PH_3302_08_ONN W153.07 BOOL  ; PH. MB FEED IN CONFIRM on
PH_3302_09_OFF W154.09 BOOL  ; PH. WORK FULL off
PH_3302_09_ON W151.09 BOOL  ; PH. WORK FULL on
PH_3302_10_OFF W154.10 BOOL  ; PH.TRANSFER STATION DIAPH SIDE CONFIRM off
PH_3302_10_ON W151.10 BOOL  ; PH.TRANSFER STATION DIAPH SIDE CONFIRM on
PH_3302_11_OFF W154.11 BOOL  ; PH.TRANSFER STATION DIAPH WORK CONFIRM off
PH_3302_11_ON W151.11 BOOL  ; PH.TRANSFER STATION DIAPH WORK CONFIRM on
PH_3302_12_OFF W154.12 BOOL  ; PH.TRANSFER STATION M&B WORK CONFIRM off
PH_3302_12_ON W151.12 BOOL  ; PH.TRANSFER STATION M&B WORK CONFIRM on
PH_3302_13_OFF W154.13 BOOL  ; PH. M&B LOADER WORK CONF 1 off
PH_3302_13_ON W151.13 BOOL  ; PH. M&B LOADER WORK CONF 1 on
PH_3302_14_OFF W154.14 BOOL  ; PH. M&B LOADER WORK CONF 2 off
PH_3302_14_ON W151.14 BOOL  ; PH. M&B LOADER WORK CONF 2 on
PH_3302_15_OFF W154.15 BOOL  ; PH. WORK IN ROTATE UNIT CONFIRM off
PH_3302_15_ON W151.15 BOOL  ; PH. WORK IN ROTATE UNIT CONFIRM on
PH_3304_08_OFF W156.08 BOOL  ; PH. WORK ROTATE PRE-END CONFIRM of
PH_3304_08_ON W153.08 BOOL  ; PH. WORK ROTATE PRE-END CONFIRM on
PH_3304_09_OFF W156.09 BOOL  ; PH. TEMINAL IN POSITION CONFIRM off
PH_3304_09_ON W153.09 BOOL  ; PH. TEMINAL IN POSITION CONFIRM on
PH_3304_10_OFF W156.10 BOOL  ; PH. WORK DIAPH LOAD IN CONFIRM off
PH_3304_10_ON W153.10 BOOL  ; PH. WORK DIAPH LOAD IN CONFIRM on
PH_3304_11_OFF W156.11 BOOL  ; PH.STATION DIAPH VACCUM CONFIRM off
PH_3304_11_ON W153.11 BOOL  ; PH.STATION DIAPH VACCUM CONFIRM on
PH_3304_12_OFF W156.12 BOOL  ; PH.STATION BUFFER DIAPH CONFIRM off
PH_3304_12_ON W153.12 BOOL  ; PH.STATION BUFFER DIAPH CONFIRM on
PH_3304_13_OFF W156.13 BOOL  ; PH. WORK NG CONFIRM off
PH_3304_13_ON W153.13 BOOL  ; PH. WORK NG CONFIRM on
PH_3304_14_OFF W156.14 BOOL  ; PH. WORK OK CONFIRM off
PH_3304_14_ON W153.14 BOOL  ; PH. WORK OK CONFIRM on
PRESSURE_NORMAL W100.01 BOOL  ; AIR SOURCE CONFIRM.
PSD W509 WORD[3]  ; SystemArea
SAFETY_DOOR W100.08 BOOL  ; CR.MACHINR DOOR CONFIRM
SHUTTER_DOOR_IN W100.11 BOOL  ; CR.SHUTTER DOOR IN CONFIRM
SHUTTER_DOOR_OUT W100.10 BOOL  ; CR.SHUTTER DOOR OUT CONFIRM
SS_AUTO W100.02 BOOL  ; AUTO.IND.(AUTO=on) On
SS_IND W200.02 BOOL  ; AUTO.IND.(AUTO=on) off
Stopwatch E0_4 UINT
Stopwatch_2 E0_5 UINT
TEACH_ON W100.07 BOOL  ; CR.TEACHING ON
sim_mch E0_3.10 BOOL

## Program P10_MAIN (cyclic task 0)
; STATION STATION CHECK
Local symbols
ALT36 T3042 TIMER
ALT37 T3000 TIMER
Disch_Command_P11 E0_3.11 BOOL
Disch_compl_aux E0_3.12 BOOL
Disch_compl_aux2 E0_3.13 BOOL
E0_3201_06 E0_46.04 BOOL  ; pin down
GB010_069 E0_3.14 BOOL  ; Homepos for discharge
Homepos_after_disch E0_3.15 BOOL
LB2341 E0_45.15 BOOL  ; PB trial mode
LB3421 E0_46.06 BOOL  ; GP1 takeout fault
LB523 E0_6.00 BOOL  ; Homeps 1 cond
LB5342 E0_45.14 BOOL  ; trigger ct
LB5431 E0_45.13 BOOL  ; trigger ct history
LD312 E0_48 UINT
LT028 T3033 TIMER
LT213 T3001 TIMER
LT214 T3002 TIMER
LT215 T3003 TIMER
LT216 T3004 TIMER
LT217 T3005 TIMER
LT2341 T3038 TIMER
LT321 T3006 TIMER  ; disch cancel
LT323 T3022 TIMER
LT324 T3021 TIMER
LT4014 T3007 TIMER
LT40505 T3008 TIMER
LT476 T3009 TIMER
LT567 T3031 TIMER
LT645 T3010 TIMER
LT765 T3034 TIMER  ; timeout positioning
LT976 T3011 TIMER
Machine_stop E0_6.01 BOOL
NOP E0_6.02 BOOL
Simulation_MCH E0_6.03 BOOL
disch_cancel E0_47.10 BOOL
nunggu_PSU E0_6.04 BOOL
rewrwe T3012 TIMER  ; Work On-> NG judge
tstt E0_45.12 BOOL

### Section MAIN

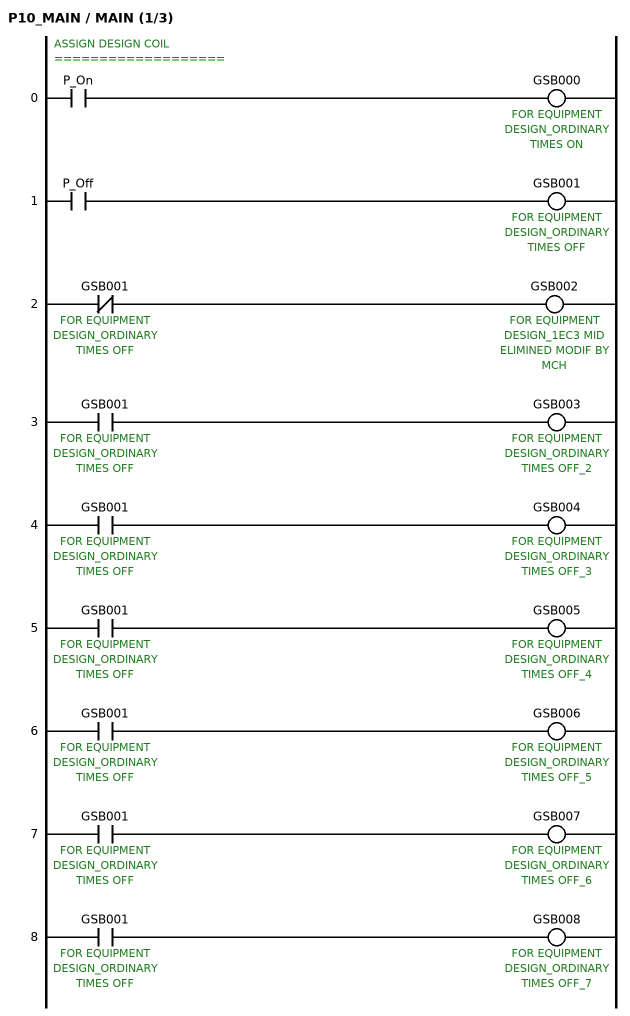
; rung 0: ASSIGN DESIGN COIL / ===================
LD P_On
OUT GSB000  ; FOR EQUIPMENT DESIGN_ORDINARY TIMES ON
; rung 1
LD P_Off
OUT GSB001  ; FOR EQUIPMENT DESIGN_ORDINARY TIMES OFF
; rung 2
LDNOT GSB001  ; FOR EQUIPMENT DESIGN_ORDINARY TIMES OFF
OUT GSB002  ; FOR EQUIPMENT DESIGN_1EC3 MID ELIMINED MODIF BY MCH
; rung 3
LD GSB001  ; FOR EQUIPMENT DESIGN_ORDINARY TIMES OFF
OUT GSB003  ; FOR EQUIPMENT DESIGN_ORDINARY TIMES OFF_2
; rung 4
LD GSB001  ; FOR EQUIPMENT DESIGN_ORDINARY TIMES OFF
OUT GSB004  ; FOR EQUIPMENT DESIGN_ORDINARY TIMES OFF_3
; rung 5
LD GSB001  ; FOR EQUIPMENT DESIGN_ORDINARY TIMES OFF
OUT GSB005  ; FOR EQUIPMENT DESIGN_ORDINARY TIMES OFF_4
; rung 6
LD GSB001  ; FOR EQUIPMENT DESIGN_ORDINARY TIMES OFF
OUT GSB006  ; FOR EQUIPMENT DESIGN_ORDINARY TIMES OFF_5
; rung 7
LD GSB001  ; FOR EQUIPMENT DESIGN_ORDINARY TIMES OFF
OUT GSB007  ; FOR EQUIPMENT DESIGN_ORDINARY TIMES OFF_6
; rung 8
LD GSB001  ; FOR EQUIPMENT DESIGN_ORDINARY TIMES OFF
OUT GSB008  ; FOR EQUIPMENT DESIGN_ORDINARY TIMES OFF_7

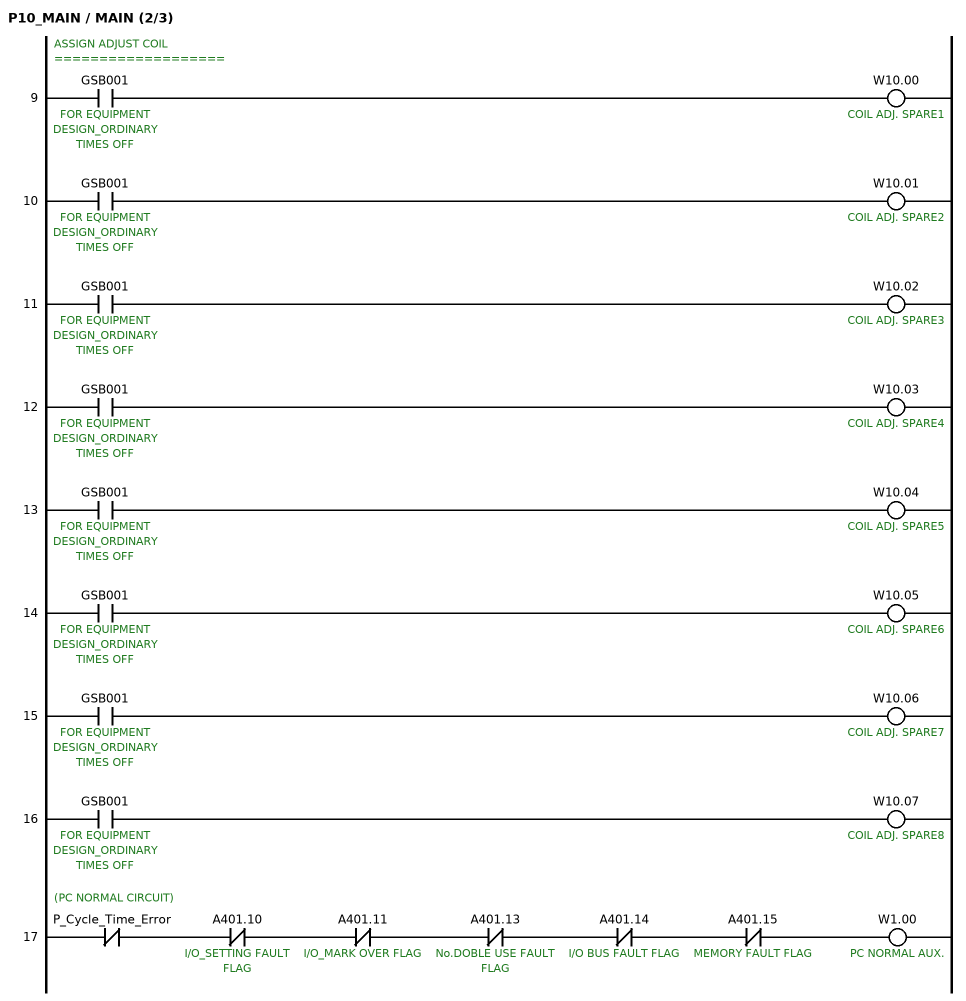
; rung 9: ASSIGN ADJUST COIL / ===================
LD GSB001  ; FOR EQUIPMENT DESIGN_ORDINARY TIMES OFF
OUT W10.00  ; COIL ADJ. SPARE1
; rung 10
LD GSB001  ; FOR EQUIPMENT DESIGN_ORDINARY TIMES OFF
OUT W10.01  ; COIL ADJ. SPARE2
; rung 11
LD GSB001  ; FOR EQUIPMENT DESIGN_ORDINARY TIMES OFF
OUT W10.02  ; COIL ADJ. SPARE3
; rung 12
LD GSB001  ; FOR EQUIPMENT DESIGN_ORDINARY TIMES OFF
OUT W10.03  ; COIL ADJ. SPARE4
; rung 13
LD GSB001  ; FOR EQUIPMENT DESIGN_ORDINARY TIMES OFF
OUT W10.04  ; COIL ADJ. SPARE5
; rung 14
LD GSB001  ; FOR EQUIPMENT DESIGN_ORDINARY TIMES OFF
OUT W10.05  ; COIL ADJ. SPARE6
; rung 15
LD GSB001  ; FOR EQUIPMENT DESIGN_ORDINARY TIMES OFF
OUT W10.06  ; COIL ADJ. SPARE7
; rung 16
LD GSB001  ; FOR EQUIPMENT DESIGN_ORDINARY TIMES OFF
OUT W10.07  ; COIL ADJ. SPARE8
; rung 17: (PC NORMAL CIRCUIT)
LDNOT P_Cycle_Time_Error
ANDNOT A401.10  ; I/O_SETTING FAULT FLAG
ANDNOT A401.11  ; I/O_MARK OVER FLAG
ANDNOT A401.13  ; No.DOBLE USE FAULT FLAG
ANDNOT A401.14  ; I/O BUS FAULT FLAG
ANDNOT A401.15  ; MEMORY FAULT FLAG
OUT W1.00  ; PC NORMAL AUX.

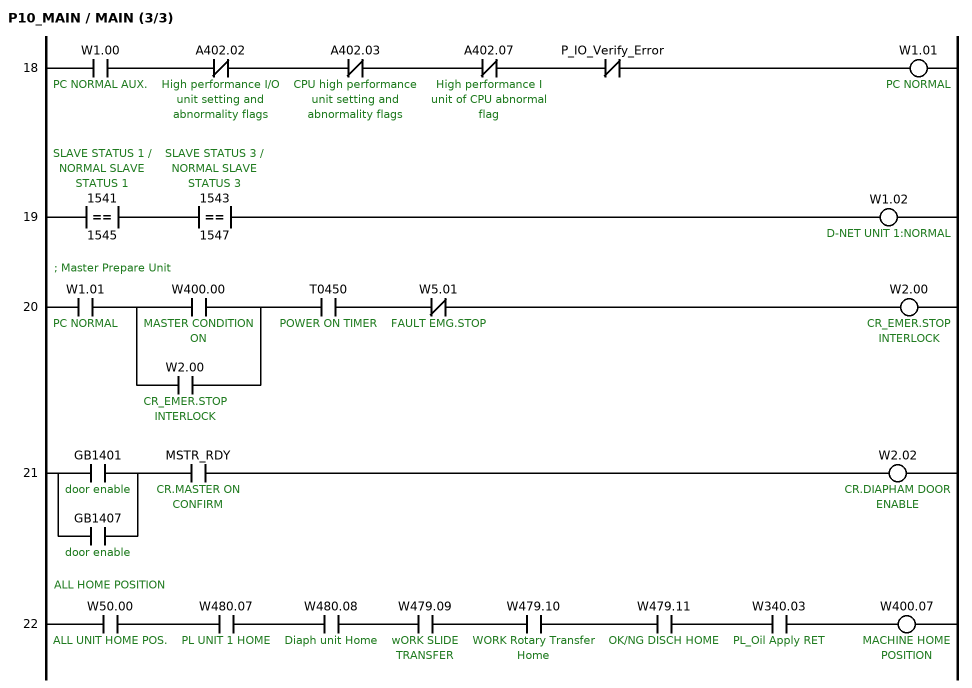
; rung 18
LD W1.00  ; PC NORMAL AUX.
ANDNOT A402.02  ; High performance I/O unit setting and abnormality flags
ANDNOT A402.03  ; CPU high performance unit setting and abnormality flags
ANDNOT A402.07  ; High performance I unit of CPU abnormal flag
ANDNOT P_IO_Verify_Error
OUT W1.01  ; PC NORMAL
; rung 19
LD=L(301) 1541 1545  ; SLAVE STATUS 1, NORMAL SLAVE STATUS 1
AND=L(301) 1543 1547  ; SLAVE STATUS 3, NORMAL SLAVE STATUS 3
OUT W1.02  ; D-NET UNIT 1:NORMAL
; rung 20: ; Master Prepare Unit
LD W1.01  ; PC NORMAL
LD W400.00  ; MASTER CONDITION ON
OR W2.00  ; CR_EMER.STOP INTERLOCK
ANDLD
AND T0450  ; POWER ON TIMER
ANDNOT W5.01  ; FAULT EMG.STOP
OUT W2.00  ; CR_EMER.STOP INTERLOCK
; rung 21
LD GB1401  ; door enable
OR GB1407  ; door enable
AND MSTR_RDY  ; CR.MASTER ON CONFIRM
OUT W2.02  ; CR.DIAPHAM DOOR ENABLE
; rung 22: ALL HOME POSITION
LD W50.00  ; ALL UNIT HOME POS.
AND W480.07  ; PL UNIT 1 HOME
AND W480.08  ; Diaph unit Home
AND W479.09  ; wORK SLIDE TRANSFER
AND W479.10  ; WORK Rotary Transfer Home
AND W479.11  ; OK/NG DISCH HOME
AND W340.03  ; PL_Oil Apply RET
OUT W400.07  ; MACHINE HOME POSITION

### Section FAULT

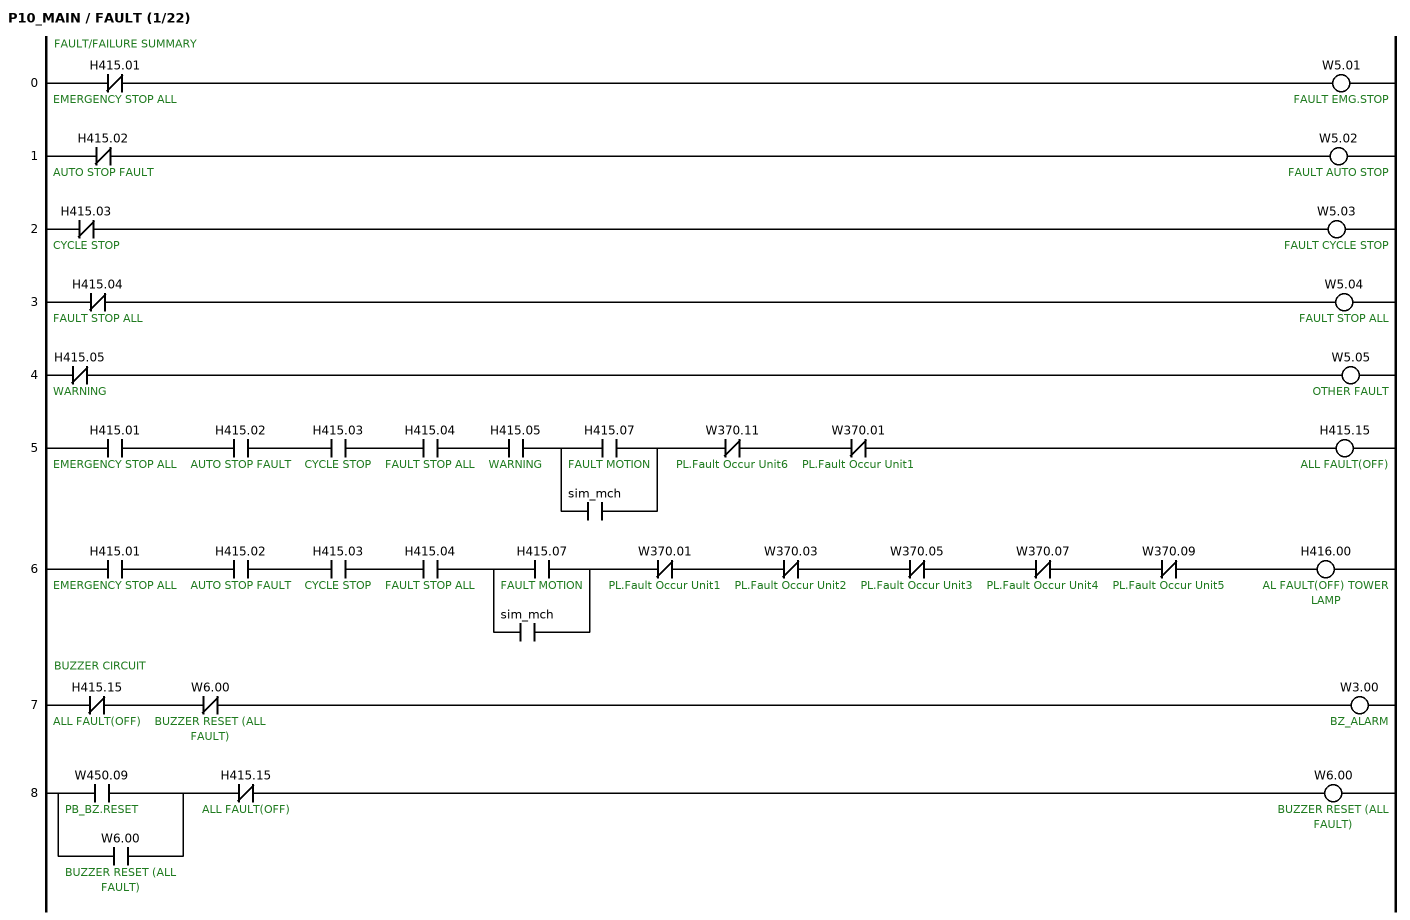
; rung 0: FAULT/FAILURE SUMMARY
LDNOT H415.01  ; EMERGENCY STOP ALL
OUT W5.01  ; FAULT EMG.STOP
; rung 1
LDNOT H415.02  ; AUTO STOP FAULT
OUT W5.02  ; FAULT AUTO STOP
; rung 2
LDNOT H415.03  ; CYCLE STOP
OUT W5.03  ; FAULT CYCLE STOP
; rung 3
LDNOT H415.04  ; FAULT STOP ALL
OUT W5.04  ; FAULT STOP ALL
; rung 4
LDNOT H415.05  ; WARNING
OUT W5.05  ; OTHER FAULT
; rung 5
LD H415.01  ; EMERGENCY STOP ALL
AND H415.02  ; AUTO STOP FAULT
AND H415.03  ; CYCLE STOP
AND H415.04  ; FAULT STOP ALL
AND H415.05  ; WARNING
LD H415.07  ; FAULT MOTION
OR sim_mch
ANDLD
ANDNOT W370.11  ; PL.Fault Occur Unit6
ANDNOT W370.01  ; PL.Fault Occur Unit1
OUT H415.15  ; ALL FAULT(OFF)
; rung 6
LD H415.01  ; EMERGENCY STOP ALL
AND H415.02  ; AUTO STOP FAULT
AND H415.03  ; CYCLE STOP
AND H415.04  ; FAULT STOP ALL
LD H415.07  ; FAULT MOTION
OR sim_mch
ANDLD
ANDNOT W370.01  ; PL.Fault Occur Unit1
ANDNOT W370.03  ; PL.Fault Occur Unit2
ANDNOT W370.05  ; PL.Fault Occur Unit3
ANDNOT W370.07  ; PL.Fault Occur Unit4
ANDNOT W370.09  ; PL.Fault Occur Unit5
OUT H416.00  ; AL FAULT(OFF) TOWER LAMP
; rung 7: BUZZER CIRCUIT
LDNOT H415.15  ; ALL FAULT(OFF)
ANDNOT W6.00  ; BUZZER RESET (ALL FAULT)
OUT W3.00  ; BZ_ALARM
; rung 8
LD W450.09  ; PB_BZ.RESET
OR W6.00  ; BUZZER RESET (ALL FAULT)
ANDNOT H415.15  ; ALL FAULT(OFF)
OUT W6.00  ; BUZZER RESET (ALL FAULT)

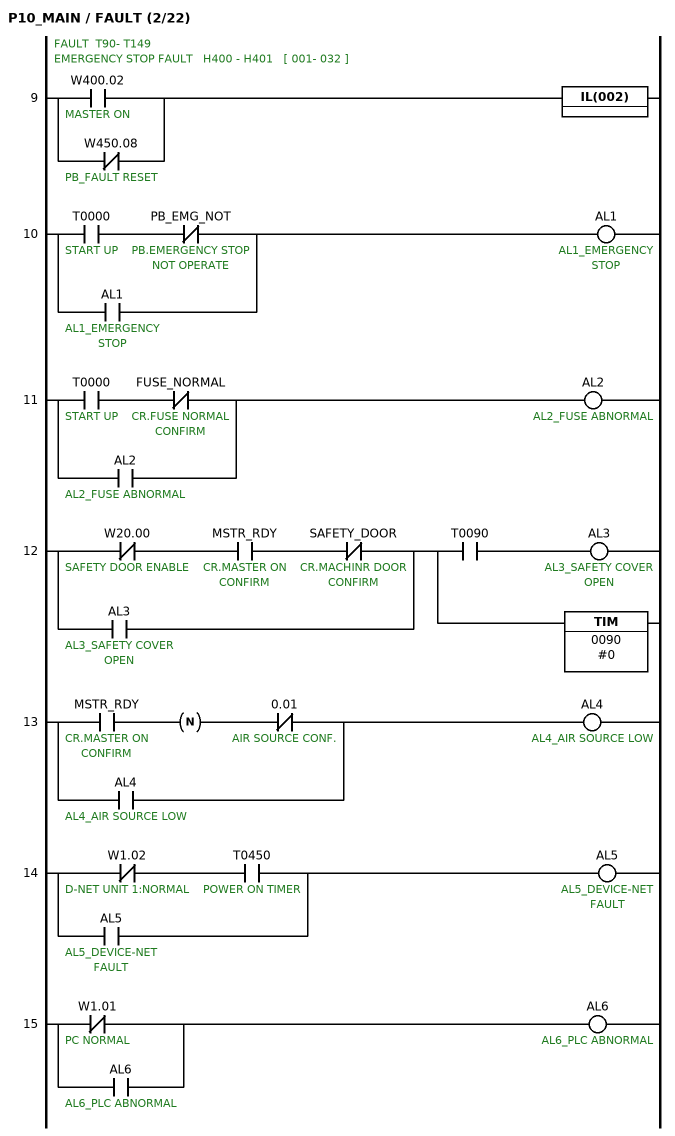
; rung 9: FAULT  T90- T149 / EMERGENCY STOP FAULT   H400 - H401   [ 001- 032 ]
LD W400.02  ; MASTER ON
ORNOT W450.08  ; PB_FAULT RESET
IL(002)
; rung 10
LD T0000  ; START UP
ANDNOT PB_EMG_NOT  ; PB.EMERGENCY STOP NOT OPERATE
OR AL1  ; AL1_EMERGENCY STOP
OUT AL1  ; AL1_EMERGENCY STOP
; rung 11
LD T0000  ; START UP
ANDNOT FUSE_NORMAL  ; CR.FUSE NORMAL CONFIRM
OR AL2  ; AL2_FUSE ABNORMAL
OUT AL2  ; AL2_FUSE ABNORMAL
; rung 12
LDNOT W20.00  ; SAFETY DOOR ENABLE
AND MSTR_RDY  ; CR.MASTER ON CONFIRM
ANDNOT SAFETY_DOOR  ; CR.MACHINR DOOR CONFIRM
OR AL3  ; AL3_SAFETY COVER OPEN
OUT TR0
AND T0090
OUT AL3  ; AL3_SAFETY COVER OPEN
LD TR0
TIM 0090 #0
; rung 13
LD MSTR_RDY  ; CR.MASTER ON CONFIRM
DOWN(522)
ANDNOT 0.01  ; AIR SOURCE CONF.
OR AL4  ; AL4_AIR SOURCE LOW
OUT AL4  ; AL4_AIR SOURCE LOW
; rung 14
LDNOT W1.02  ; D-NET UNIT 1:NORMAL
AND T0450  ; POWER ON TIMER
OR AL5  ; AL5_DEVICE-NET FAULT
OUT AL5  ; AL5_DEVICE-NET FAULT
; rung 15
LDNOT W1.01  ; PC NORMAL
OR AL6  ; AL6_PLC ABNORMAL
OUT AL6  ; AL6_PLC ABNORMAL

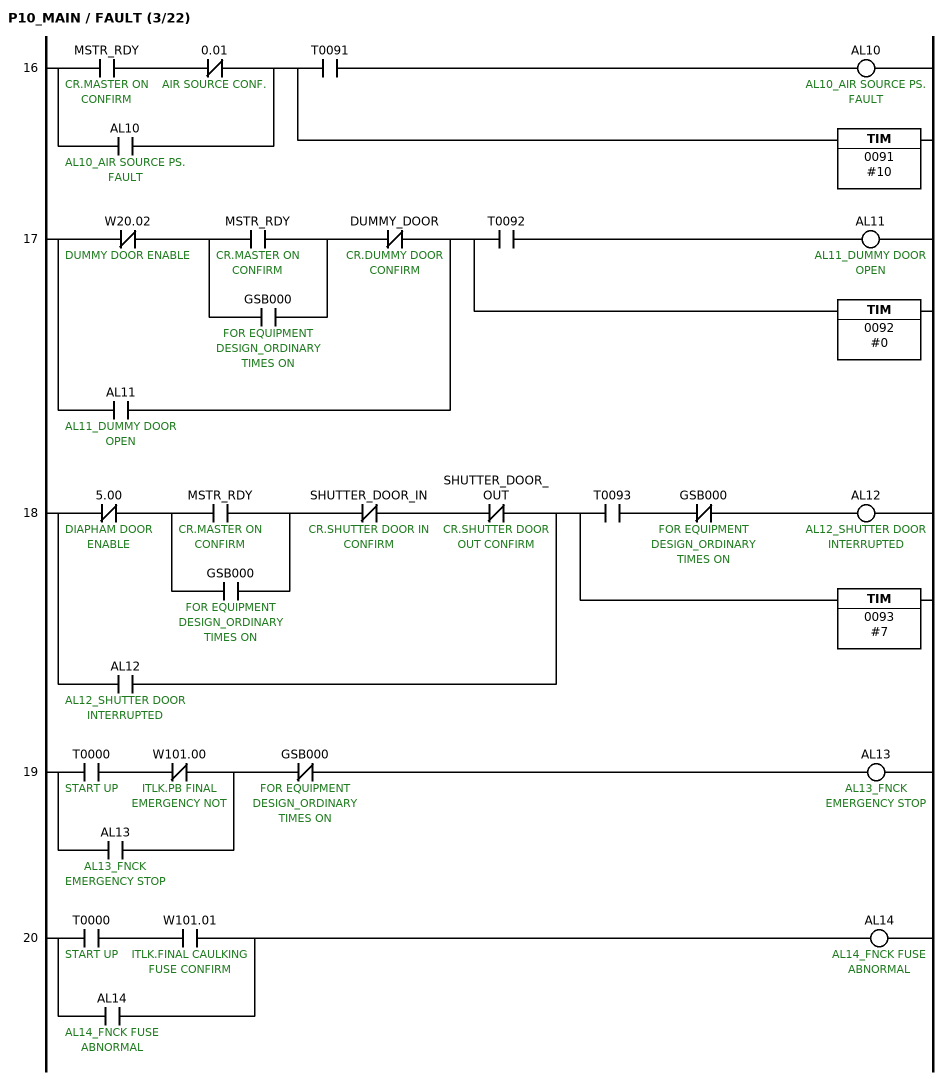
; rung 16
LD MSTR_RDY  ; CR.MASTER ON CONFIRM
ANDNOT 0.01  ; AIR SOURCE CONF.
OR AL10  ; AL10_AIR SOURCE PS. FAULT
OUT TR0
AND T0091
OUT AL10  ; AL10_AIR SOURCE PS. FAULT
LD TR0
TIM 0091 #10
; rung 17
LDNOT W20.02  ; DUMMY DOOR ENABLE
LD MSTR_RDY  ; CR.MASTER ON CONFIRM
OR GSB000  ; FOR EQUIPMENT DESIGN_ORDINARY TIMES ON
ANDLD
ANDNOT DUMMY_DOOR  ; CR.DUMMY DOOR CONFIRM
OR AL11  ; AL11_DUMMY DOOR OPEN
OUT TR0
AND T0092
OUT AL11  ; AL11_DUMMY DOOR OPEN
LD TR0
TIM 0092 #0
; rung 18
LDNOT 5.00  ; DIAPHAM DOOR ENABLE
LD MSTR_RDY  ; CR.MASTER ON CONFIRM
OR GSB000  ; FOR EQUIPMENT DESIGN_ORDINARY TIMES ON
ANDLD
ANDNOT SHUTTER_DOOR_IN  ; CR.SHUTTER DOOR IN CONFIRM
ANDNOT SHUTTER_DOOR_OUT  ; CR.SHUTTER DOOR OUT CONFIRM
OR AL12  ; AL12_SHUTTER DOOR INTERRUPTED
OUT TR0
AND T0093
ANDNOT GSB000  ; FOR EQUIPMENT DESIGN_ORDINARY TIMES ON
OUT AL12  ; AL12_SHUTTER DOOR INTERRUPTED
LD TR0
TIM 0093 #7
; rung 19
LD T0000  ; START UP
ANDNOT W101.00  ; ITLK.PB FINAL EMERGENCY NOT
OR AL13  ; AL13_FNCK EMERGENCY STOP
ANDNOT GSB000  ; FOR EQUIPMENT DESIGN_ORDINARY TIMES ON
OUT AL13  ; AL13_FNCK EMERGENCY STOP
; rung 20
LD T0000  ; START UP
AND W101.01  ; ITLK.FINAL CAULKING FUSE CONFIRM
OR AL14  ; AL14_FNCK FUSE ABNORMAL
OUT AL14  ; AL14_FNCK FUSE ABNORMAL

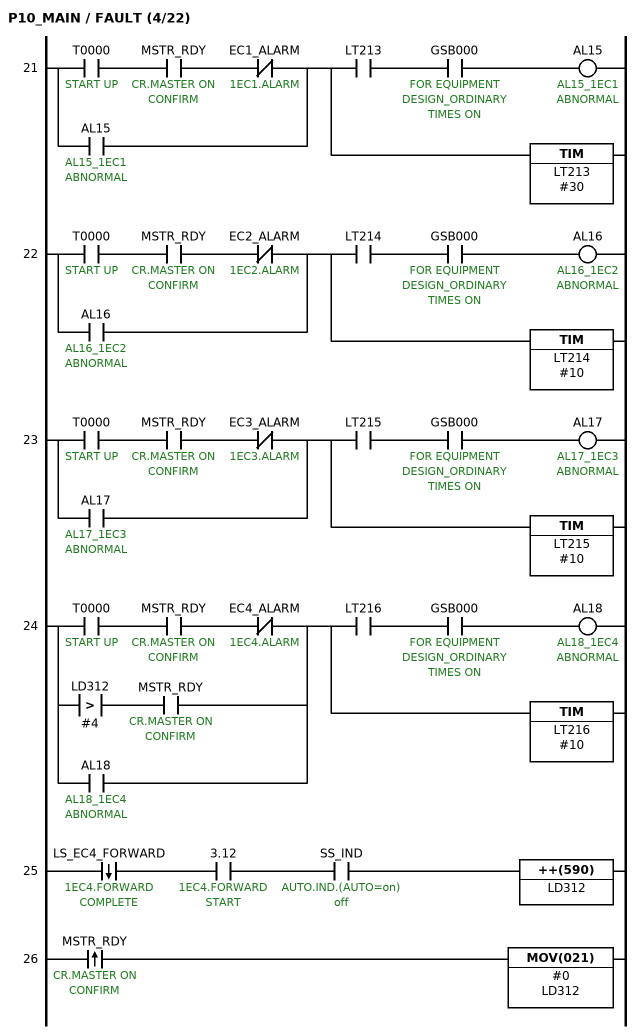
; rung 21
LD T0000  ; START UP
AND MSTR_RDY  ; CR.MASTER ON CONFIRM
ANDNOT EC1_ALARM  ; 1EC1.ALARM
OR AL15  ; AL15_1EC1 ABNORMAL
OUT TR0
AND LT213
AND GSB000  ; FOR EQUIPMENT DESIGN_ORDINARY TIMES ON
OUT AL15  ; AL15_1EC1 ABNORMAL
LD TR0
TIM LT213 #30
; rung 22
LD T0000  ; START UP
AND MSTR_RDY  ; CR.MASTER ON CONFIRM
ANDNOT EC2_ALARM  ; 1EC2.ALARM
OR AL16  ; AL16_1EC2 ABNORMAL
OUT TR0
AND LT214
AND GSB000  ; FOR EQUIPMENT DESIGN_ORDINARY TIMES ON
OUT AL16  ; AL16_1EC2 ABNORMAL
LD TR0
TIM LT214 #10
; rung 23
LD T0000  ; START UP
AND MSTR_RDY  ; CR.MASTER ON CONFIRM
ANDNOT EC3_ALARM  ; 1EC3.ALARM
OR AL17  ; AL17_1EC3 ABNORMAL
OUT TR0
AND LT215
AND GSB000  ; FOR EQUIPMENT DESIGN_ORDINARY TIMES ON
OUT AL17  ; AL17_1EC3 ABNORMAL
LD TR0
TIM LT215 #10
; rung 24
LD T0000  ; START UP
AND MSTR_RDY  ; CR.MASTER ON CONFIRM
ANDNOT EC4_ALARM  ; 1EC4.ALARM
LD>(320) LD312 #4
AND MSTR_RDY  ; CR.MASTER ON CONFIRM
ORLD
OR AL18  ; AL18_1EC4 ABNORMAL
OUT TR0
AND LT216
AND GSB000  ; FOR EQUIPMENT DESIGN_ORDINARY TIMES ON
OUT AL18  ; AL18_1EC4 ABNORMAL
LD TR0
TIM LT216 #10
; rung 25
%LD LS_EC4_FORWARD  ; 1EC4.FORWARD COMPLETE
AND 3.12  ; 1EC4.FORWARD START
AND SS_IND  ; AUTO.IND.(AUTO=on) off
++(590) LD312
; rung 26
@LD MSTR_RDY  ; CR.MASTER ON CONFIRM
MOV(021) #0 LD312

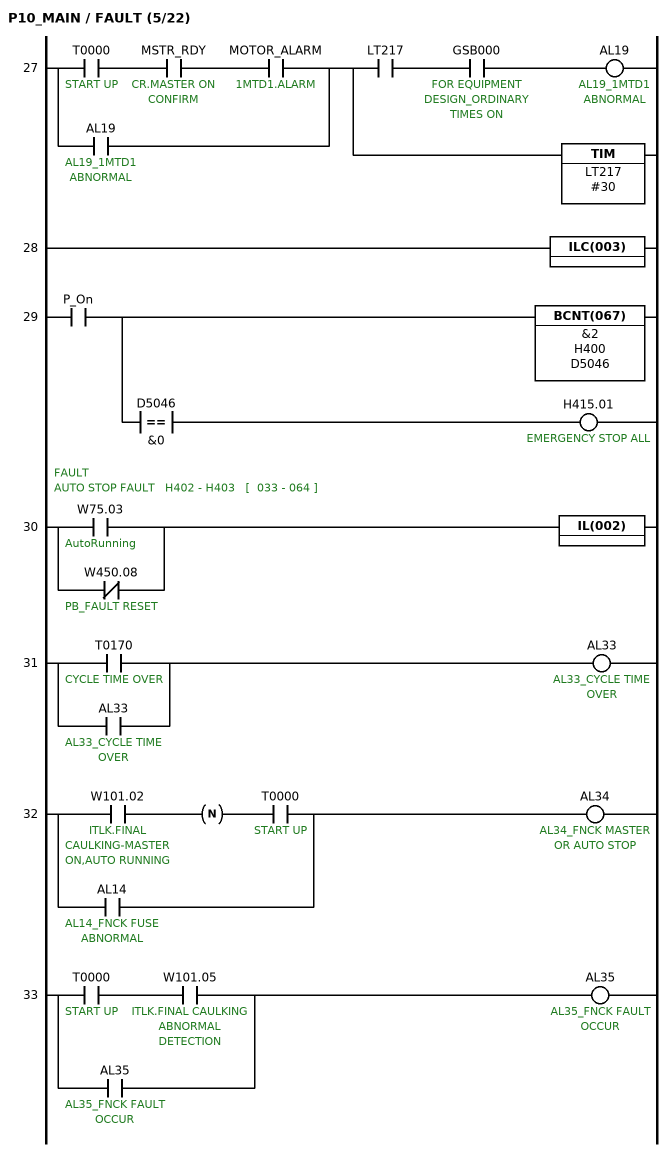
; rung 27
LD T0000  ; START UP
AND MSTR_RDY  ; CR.MASTER ON CONFIRM
AND MOTOR_ALARM  ; 1MTD1.ALARM
OR AL19  ; AL19_1MTD1 ABNORMAL
OUT TR0
AND LT217
AND GSB000  ; FOR EQUIPMENT DESIGN_ORDINARY TIMES ON
OUT AL19  ; AL19_1MTD1 ABNORMAL
LD TR0
TIM LT217 #30
; rung 28
ILC(003)
; rung 29
LD P_On
BCNT(067) &2 H400 D5046
AND=(300) D5046 &0
OUT H415.01  ; EMERGENCY STOP ALL
; rung 30: FAULT / AUTO STOP FAULT   H402 - H403   [  033 - 064 ]
LD W75.03  ; AutoRunning
ORNOT W450.08  ; PB_FAULT RESET
IL(002)
; rung 31
LD T0170  ; CYCLE TIME OVER
OR AL33  ; AL33_CYCLE TIME OVER
OUT AL33  ; AL33_CYCLE TIME OVER
; rung 32
LD W101.02  ; ITLK.FINAL CAULKING-MASTER ON,AUTO RUNNING
DOWN(522)
AND T0000  ; START UP
OR AL14  ; AL14_FNCK FUSE ABNORMAL
OUT AL34  ; AL34_FNCK MASTER OR AUTO STOP
; rung 33
LD T0000  ; START UP
AND W101.05  ; ITLK.FINAL CAULKING ABNORMAL DETECTION
OR AL35  ; AL35_FNCK FAULT OCCUR
OUT AL35  ; AL35_FNCK FAULT OCCUR

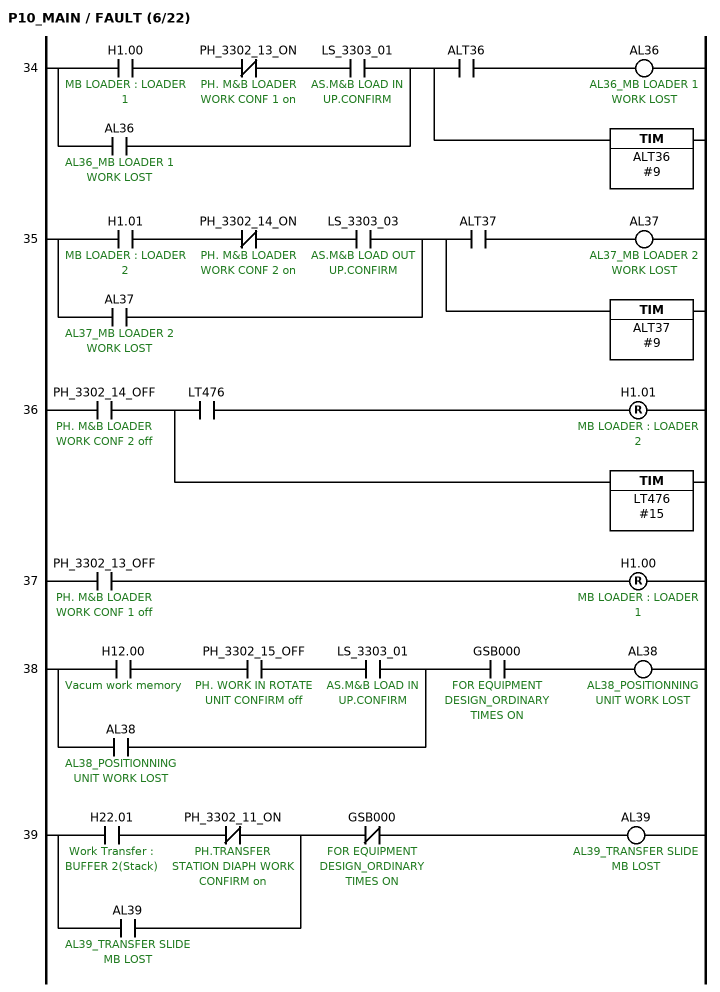
; rung 34
LD H1.00  ; MB LOADER : LOADER 1
ANDNOT PH_3302_13_ON  ; PH. M&B LOADER WORK CONF 1 on
AND LS_3303_01  ; AS.M&B LOAD IN UP.CONFIRM
OR AL36  ; AL36_MB LOADER 1 WORK LOST
OUT TR0
AND ALT36
OUT AL36  ; AL36_MB LOADER 1 WORK LOST
LD TR0
TIM ALT36 #9
; rung 35
LD H1.01  ; MB LOADER : LOADER 2
ANDNOT PH_3302_14_ON  ; PH. M&B LOADER WORK CONF 2 on
AND LS_3303_03  ; AS.M&B LOAD OUT UP.CONFIRM
OR AL37  ; AL37_MB LOADER 2 WORK LOST
OUT TR0
AND ALT37
OUT AL37  ; AL37_MB LOADER 2 WORK LOST
LD TR0
TIM ALT37 #9
; rung 36
LD PH_3302_14_OFF  ; PH. M&B LOADER WORK CONF 2 off
OUT TR0
AND LT476
RSET H1.01  ; MB LOADER : LOADER 2
LD TR0
TIM LT476 #15
; rung 37
LD PH_3302_13_OFF  ; PH. M&B LOADER WORK CONF 1 off
RSET H1.00  ; MB LOADER : LOADER 1
; rung 38
LD H12.00  ; Vacum work memory
AND PH_3302_15_OFF  ; PH. WORK IN ROTATE UNIT CONFIRM off
AND LS_3303_01  ; AS.M&B LOAD IN UP.CONFIRM
OR AL38  ; AL38_POSITIONNING UNIT WORK LOST
AND GSB000  ; FOR EQUIPMENT DESIGN_ORDINARY TIMES ON
OUT AL38  ; AL38_POSITIONNING UNIT WORK LOST
; rung 39
LD H22.01  ; Work Transfer : BUFFER 2(Stack)
ANDNOT PH_3302_11_ON  ; PH.TRANSFER STATION DIAPH WORK CONFIRM on
OR AL39  ; AL39_TRANSFER SLIDE MB LOST
ANDNOT GSB000  ; FOR EQUIPMENT DESIGN_ORDINARY TIMES ON
OUT AL39  ; AL39_TRANSFER SLIDE MB LOST

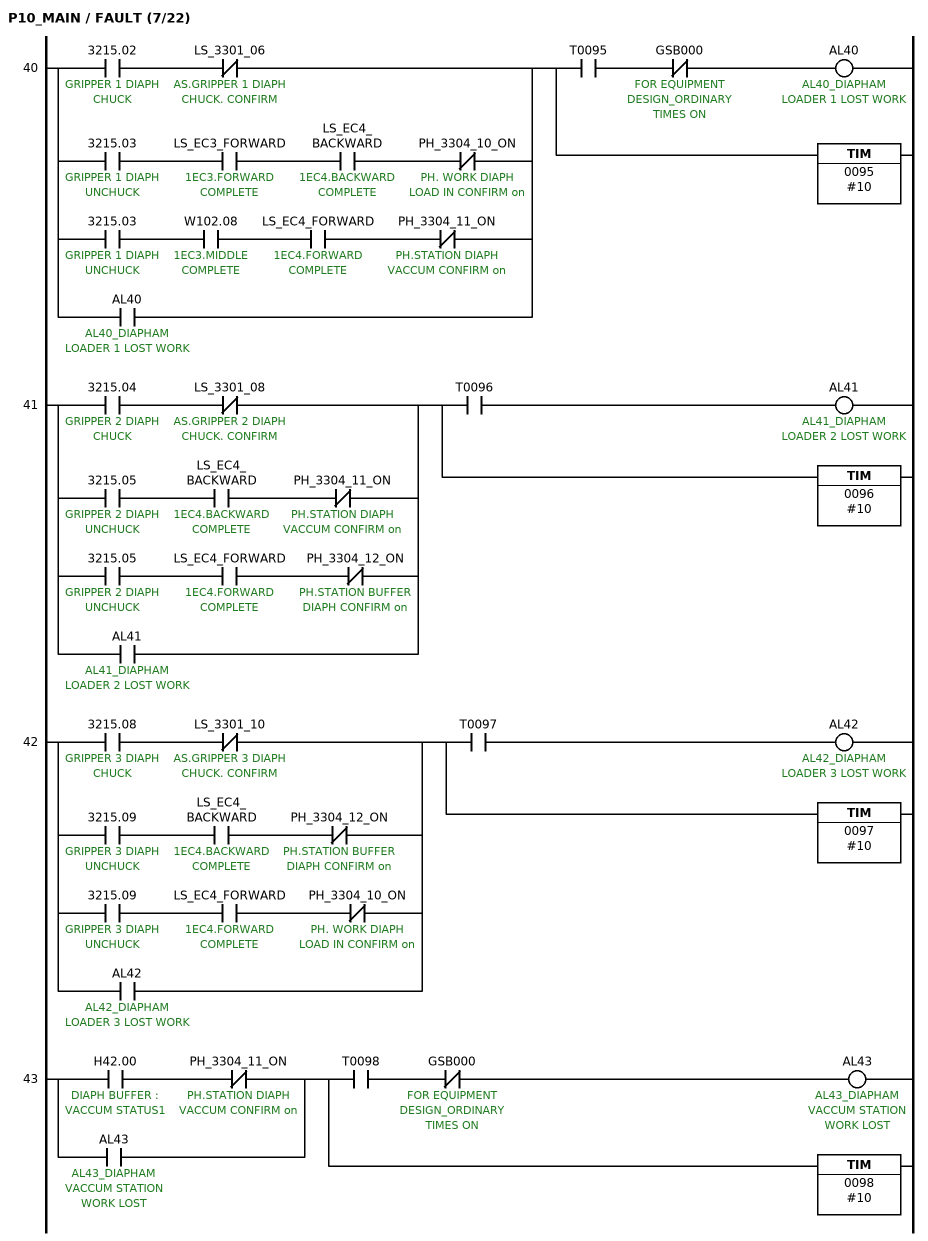
; rung 40
LD 3215.02  ; GRIPPER 1 DIAPH CHUCK
ANDNOT LS_3301_06  ; AS.GRIPPER 1 DIAPH CHUCK. CONFIRM
LD 3215.03  ; GRIPPER 1 DIAPH UNCHUCK
AND LS_EC3_FORWARD  ; 1EC3.FORWARD COMPLETE
AND LS_EC4_BACKWARD  ; 1EC4.BACKWARD COMPLETE
ANDNOT PH_3304_10_ON  ; PH. WORK DIAPH LOAD IN CONFIRM on
ORLD
LD 3215.03  ; GRIPPER 1 DIAPH UNCHUCK
AND W102.08  ; 1EC3.MIDDLE COMPLETE
AND LS_EC4_FORWARD  ; 1EC4.FORWARD COMPLETE
ANDNOT PH_3304_11_ON  ; PH.STATION DIAPH VACCUM CONFIRM on
ORLD
OR AL40  ; AL40_DIAPHAM LOADER 1 LOST WORK
OUT TR0
AND T0095
ANDNOT GSB000  ; FOR EQUIPMENT DESIGN_ORDINARY TIMES ON
OUT AL40  ; AL40_DIAPHAM LOADER 1 LOST WORK
LD TR0
TIM 0095 #10
; rung 41
LD 3215.04  ; GRIPPER 2 DIAPH CHUCK
ANDNOT LS_3301_08  ; AS.GRIPPER 2 DIAPH CHUCK. CONFIRM
LD 3215.05  ; GRIPPER 2 DIAPH UNCHUCK
AND LS_EC4_BACKWARD  ; 1EC4.BACKWARD COMPLETE
ANDNOT PH_3304_11_ON  ; PH.STATION DIAPH VACCUM CONFIRM on
ORLD
LD 3215.05  ; GRIPPER 2 DIAPH UNCHUCK
AND LS_EC4_FORWARD  ; 1EC4.FORWARD COMPLETE
ANDNOT PH_3304_12_ON  ; PH.STATION BUFFER DIAPH CONFIRM on
ORLD
OR AL41  ; AL41_DIAPHAM LOADER 2 LOST WORK
OUT TR0
AND T0096
OUT AL41  ; AL41_DIAPHAM LOADER 2 LOST WORK
LD TR0
TIM 0096 #10
; rung 42
LD 3215.08  ; GRIPPER 3 DIAPH CHUCK
ANDNOT LS_3301_10  ; AS.GRIPPER 3 DIAPH CHUCK. CONFIRM
LD 3215.09  ; GRIPPER 3 DIAPH UNCHUCK
AND LS_EC4_BACKWARD  ; 1EC4.BACKWARD COMPLETE
ANDNOT PH_3304_12_ON  ; PH.STATION BUFFER DIAPH CONFIRM on
ORLD
LD 3215.09  ; GRIPPER 3 DIAPH UNCHUCK
AND LS_EC4_FORWARD  ; 1EC4.FORWARD COMPLETE
ANDNOT PH_3304_10_ON  ; PH. WORK DIAPH LOAD IN CONFIRM on
ORLD
OR AL42  ; AL42_DIAPHAM LOADER 3 LOST WORK
OUT TR0
AND T0097
OUT AL42  ; AL42_DIAPHAM LOADER 3 LOST WORK
LD TR0
TIM 0097 #10
; rung 43
LD H42.00  ; DIAPH BUFFER : VACCUM STATUS1
ANDNOT PH_3304_11_ON  ; PH.STATION DIAPH VACCUM CONFIRM on
OR AL43  ; AL43_DIAPHAM VACCUM STATION WORK LOST
OUT TR0
AND T0098
ANDNOT GSB000  ; FOR EQUIPMENT DESIGN_ORDINARY TIMES ON
OUT AL43  ; AL43_DIAPHAM VACCUM STATION WORK LOST
LD TR0
TIM 0098 #10

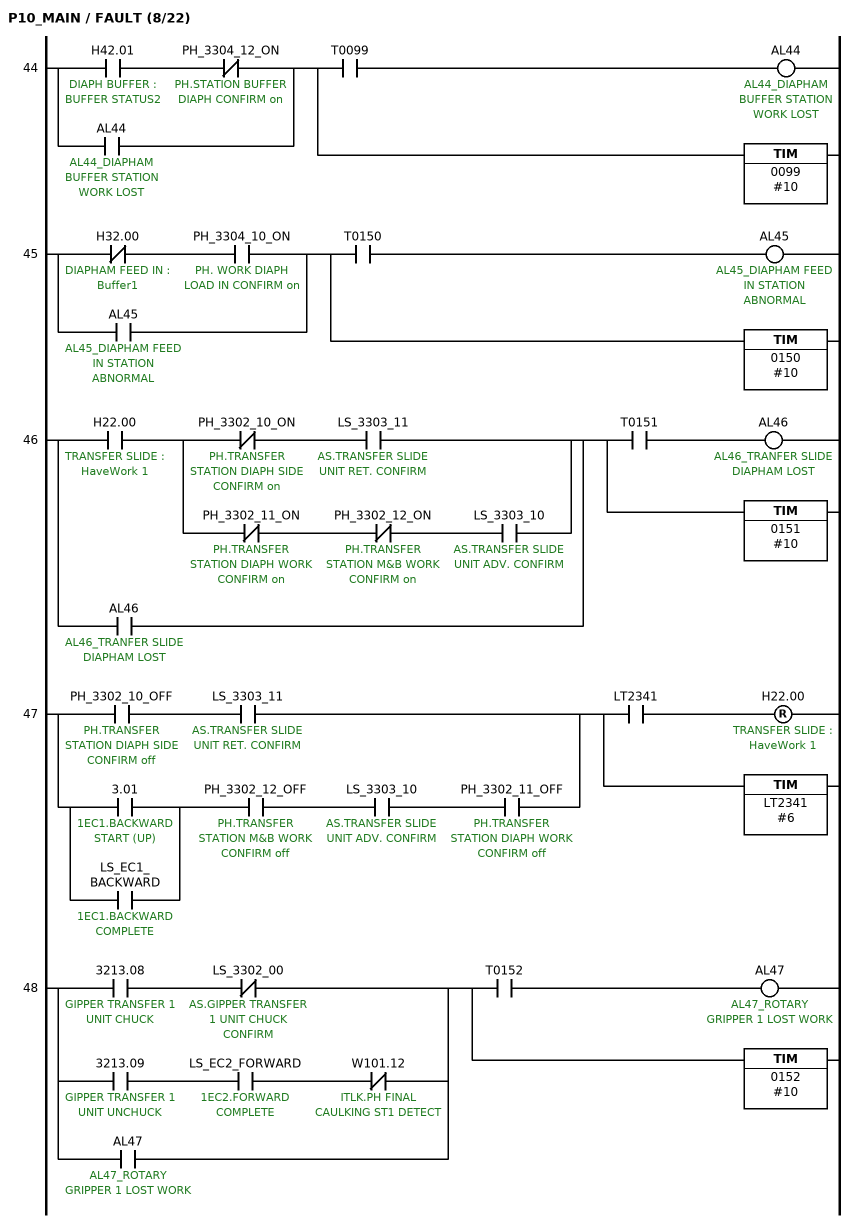
; rung 44
LD H42.01  ; DIAPH BUFFER : BUFFER STATUS2
ANDNOT PH_3304_12_ON  ; PH.STATION BUFFER DIAPH CONFIRM on
OR AL44  ; AL44_DIAPHAM BUFFER STATION WORK LOST
OUT TR0
AND T0099
OUT AL44  ; AL44_DIAPHAM BUFFER STATION WORK LOST
LD TR0
TIM 0099 #10
; rung 45
LDNOT H32.00  ; DIAPHAM FEED IN : Buffer1
AND PH_3304_10_ON  ; PH. WORK DIAPH LOAD IN CONFIRM on
OR AL45  ; AL45_DIAPHAM FEED IN STATION ABNORMAL
OUT TR0
AND T0150
OUT AL45  ; AL45_DIAPHAM FEED IN STATION ABNORMAL
LD TR0
TIM 0150 #10
; rung 46
LD H22.00  ; TRANSFER SLIDE : HaveWork 1
LDNOT PH_3302_10_ON  ; PH.TRANSFER STATION DIAPH SIDE CONFIRM on
AND LS_3303_11  ; AS.TRANSFER SLIDE UNIT RET. CONFIRM
LDNOT PH_3302_11_ON  ; PH.TRANSFER STATION DIAPH WORK CONFIRM on
ANDNOT PH_3302_12_ON  ; PH.TRANSFER STATION M&B WORK CONFIRM on
AND LS_3303_10  ; AS.TRANSFER SLIDE UNIT ADV. CONFIRM
ORLD
ANDLD
OR AL46  ; AL46_TRANFER SLIDE DIAPHAM LOST
OUT TR0
AND T0151
OUT AL46  ; AL46_TRANFER SLIDE DIAPHAM LOST
LD TR0
TIM 0151 #10
; rung 47
LD PH_3302_10_OFF  ; PH.TRANSFER STATION DIAPH SIDE CONFIRM off
AND LS_3303_11  ; AS.TRANSFER SLIDE UNIT RET. CONFIRM
LD 3.01  ; 1EC1.BACKWARD START (UP)
OR LS_EC1_BACKWARD  ; 1EC1.BACKWARD COMPLETE
AND PH_3302_12_OFF  ; PH.TRANSFER STATION M&B WORK CONFIRM off
AND LS_3303_10  ; AS.TRANSFER SLIDE UNIT ADV. CONFIRM
AND PH_3302_11_OFF  ; PH.TRANSFER STATION DIAPH WORK CONFIRM off
ORLD
OUT TR0
AND LT2341
RSET H22.00  ; TRANSFER SLIDE : HaveWork 1
LD TR0
TIM LT2341 #6
; rung 48
LD 3213.08  ; GIPPER TRANSFER 1 UNIT CHUCK
ANDNOT LS_3302_00  ; AS.GIPPER TRANSFER 1 UNIT CHUCK CONFIRM
LD 3213.09  ; GIPPER TRANSFER 1 UNIT UNCHUCK
AND LS_EC2_FORWARD  ; 1EC2.FORWARD COMPLETE
ANDNOT W101.12  ; ITLK.PH FINAL CAULKING ST1 DETECT
ORLD
OR AL47  ; AL47_ROTARY GRIPPER 1 LOST WORK
OUT TR0
AND T0152
OUT AL47  ; AL47_ROTARY GRIPPER 1 LOST WORK
LD TR0
TIM 0152 #10

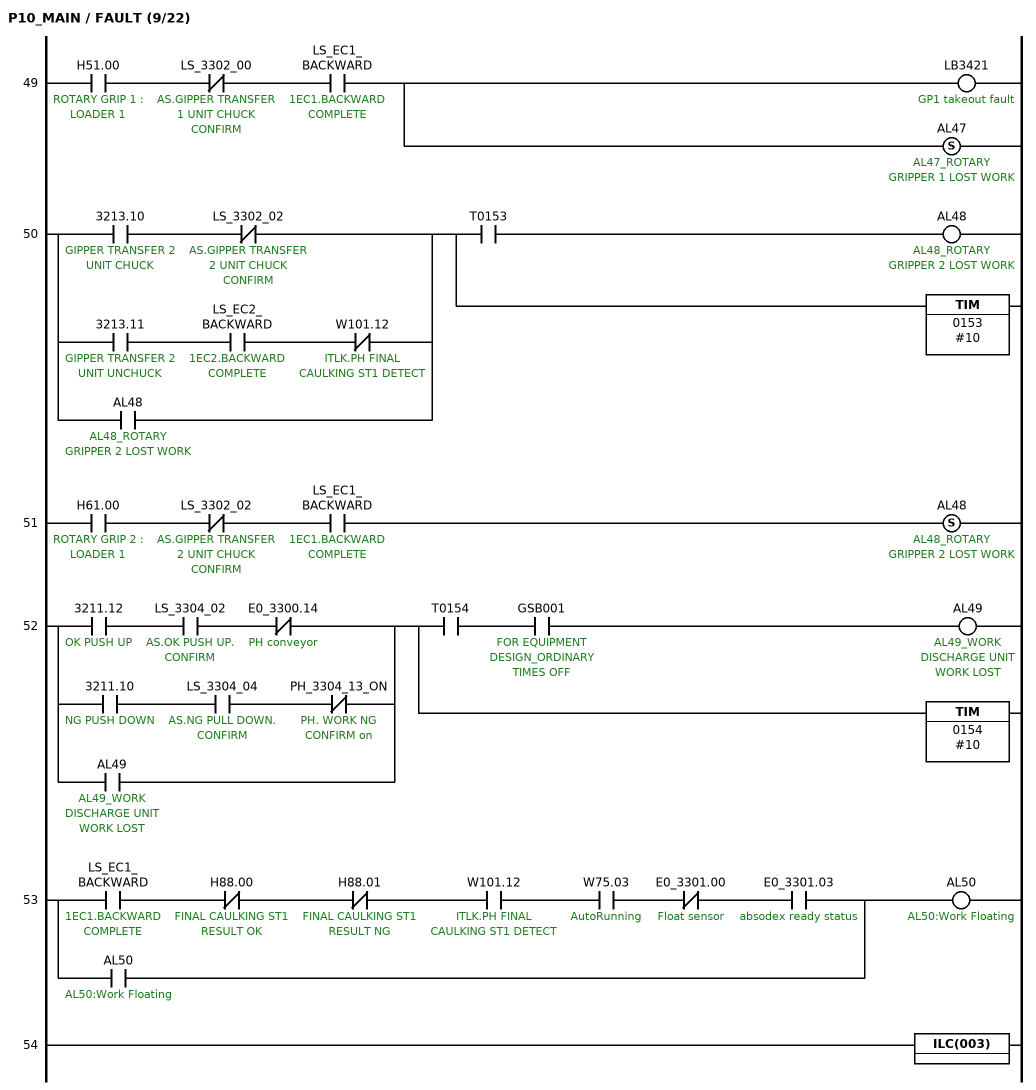
; rung 49
LD H51.00  ; ROTARY GRIP 1 : LOADER 1
ANDNOT LS_3302_00  ; AS.GIPPER TRANSFER 1 UNIT CHUCK CONFIRM
AND LS_EC1_BACKWARD  ; 1EC1.BACKWARD COMPLETE
OUT LB3421  ; GP1 takeout fault
SET AL47  ; AL47_ROTARY GRIPPER 1 LOST WORK
; rung 50
LD 3213.10  ; GIPPER TRANSFER 2 UNIT CHUCK
ANDNOT LS_3302_02  ; AS.GIPPER TRANSFER 2 UNIT CHUCK CONFIRM
LD 3213.11  ; GIPPER TRANSFER 2 UNIT UNCHUCK
AND LS_EC2_BACKWARD  ; 1EC2.BACKWARD COMPLETE
ANDNOT W101.12  ; ITLK.PH FINAL CAULKING ST1 DETECT
ORLD
OR AL48  ; AL48_ROTARY GRIPPER 2 LOST WORK
OUT TR0
AND T0153
OUT AL48  ; AL48_ROTARY GRIPPER 2 LOST WORK
LD TR0
TIM 0153 #10
; rung 51
LD H61.00  ; ROTARY GRIP 2 : LOADER 1
ANDNOT LS_3302_02  ; AS.GIPPER TRANSFER 2 UNIT CHUCK CONFIRM
AND LS_EC1_BACKWARD  ; 1EC1.BACKWARD COMPLETE
SET AL48  ; AL48_ROTARY GRIPPER 2 LOST WORK
; rung 52
LD 3211.12  ; OK PUSH UP
AND LS_3304_02  ; AS.OK PUSH UP. CONFIRM
ANDNOT E0_3300.14  ; PH conveyor
LD 3211.10  ; NG PUSH DOWN
AND LS_3304_04  ; AS.NG PULL DOWN. CONFIRM
ANDNOT PH_3304_13_ON  ; PH. WORK NG CONFIRM on
ORLD
OR AL49  ; AL49_WORK DISCHARGE UNIT WORK LOST
OUT TR0
AND T0154
AND GSB001  ; FOR EQUIPMENT DESIGN_ORDINARY TIMES OFF
OUT AL49  ; AL49_WORK DISCHARGE UNIT WORK LOST
LD TR0
TIM 0154 #10
; rung 53
LD LS_EC1_BACKWARD  ; 1EC1.BACKWARD COMPLETE
ANDNOT H88.00  ; FINAL CAULKING ST1 RESULT OK
ANDNOT H88.01  ; FINAL CAULKING ST1 RESULT NG
AND W101.12  ; ITLK.PH FINAL CAULKING ST1 DETECT
AND W75.03  ; AutoRunning
ANDNOT E0_3301.00  ; Float sensor
AND E0_3301.03  ; absodex ready status
OR AL50  ; AL50:Work Floating
OUT AL50  ; AL50:Work Floating
; rung 54
ILC(003)

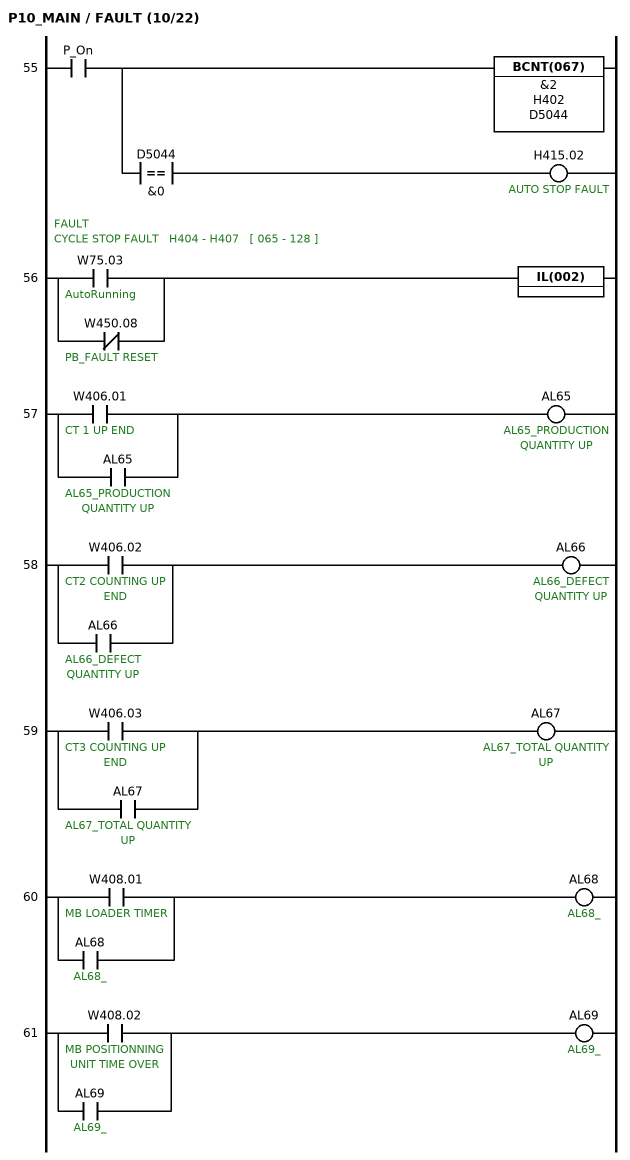
; rung 55
LD P_On
BCNT(067) &2 H402 D5044
AND=(300) D5044 &0
OUT H415.02  ; AUTO STOP FAULT
; rung 56: FAULT / CYCLE STOP FAULT   H404 - H407   [ 065 - 128 ]
LD W75.03  ; AutoRunning
ORNOT W450.08  ; PB_FAULT RESET
IL(002)
; rung 57
LD W406.01  ; CT 1 UP END
OR AL65  ; AL65_PRODUCTION QUANTITY UP
OUT AL65  ; AL65_PRODUCTION QUANTITY UP
; rung 58
LD W406.02  ; CT2 COUNTING UP END
OR AL66  ; AL66_DEFECT QUANTITY UP
OUT AL66  ; AL66_DEFECT QUANTITY UP
; rung 59
LD W406.03  ; CT3 COUNTING UP END
OR AL67  ; AL67_TOTAL QUANTITY UP
OUT AL67  ; AL67_TOTAL QUANTITY UP
; rung 60
LD W408.01  ; MB LOADER TIMER
OR AL68  ; AL68_
OUT AL68  ; AL68_
; rung 61
LD W408.02  ; MB POSITIONNING UNIT TIME OVER
OR AL69  ; AL69_
OUT AL69  ; AL69_

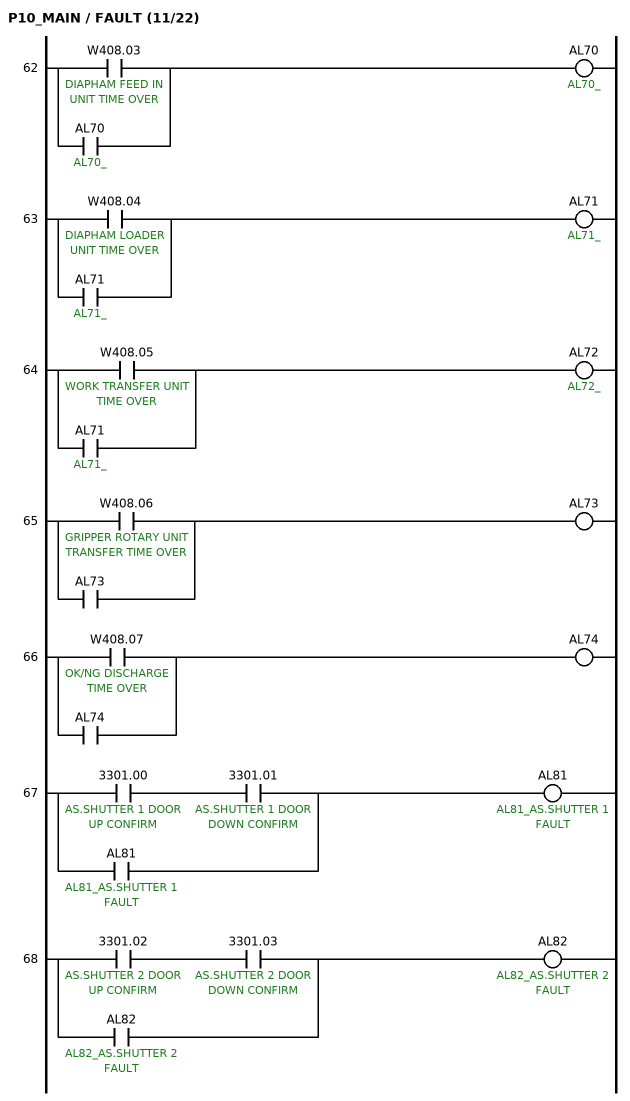
; rung 62
LD W408.03  ; DIAPHAM FEED IN UNIT TIME OVER
OR AL70  ; AL70_
OUT AL70  ; AL70_
; rung 63
LD W408.04  ; DIAPHAM LOADER UNIT TIME OVER
OR AL71  ; AL71_
OUT AL71  ; AL71_
; rung 64
LD W408.05  ; WORK TRANSFER UNIT TIME OVER
OR AL71  ; AL71_
OUT AL72  ; AL72_
; rung 65
LD W408.06  ; GRIPPER ROTARY UNIT TRANSFER TIME OVER
OR AL73
OUT AL73
; rung 66
LD W408.07  ; OK/NG DISCHARGE TIME OVER
OR AL74
OUT AL74
; rung 67
LD 3301.00  ; AS.SHUTTER 1 DOOR UP CONFIRM
AND 3301.01  ; AS.SHUTTER 1 DOOR DOWN CONFIRM
OR AL81  ; AL81_AS.SHUTTER 1 FAULT
OUT AL81  ; AL81_AS.SHUTTER 1 FAULT
; rung 68
LD 3301.02  ; AS.SHUTTER 2 DOOR UP CONFIRM
AND 3301.03  ; AS.SHUTTER 2 DOOR DOWN CONFIRM
OR AL82  ; AL82_AS.SHUTTER 2 FAULT
OUT AL82  ; AL82_AS.SHUTTER 2 FAULT

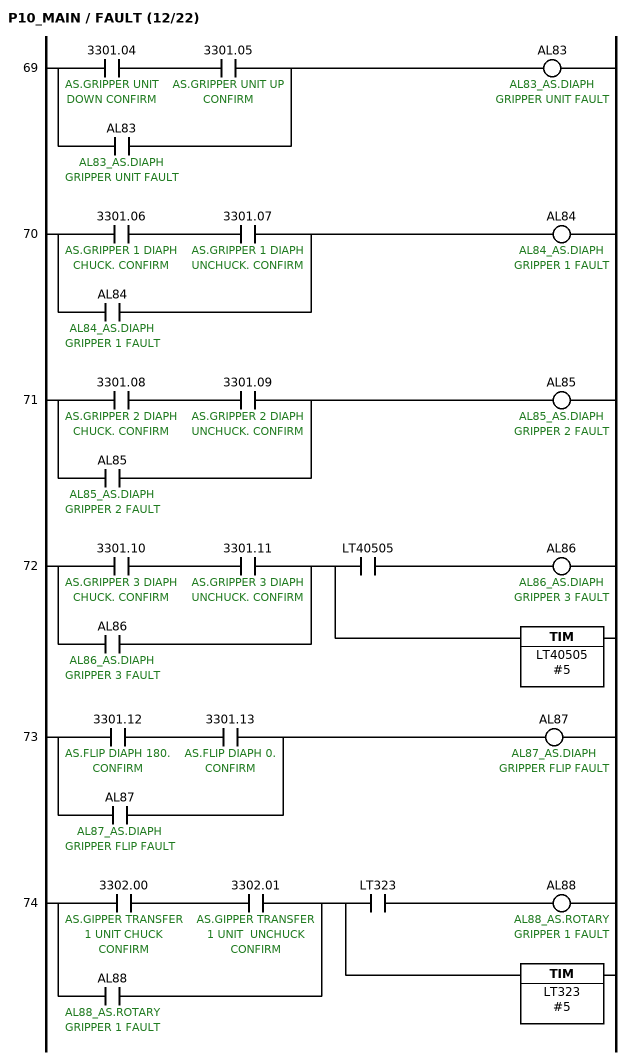
; rung 69
LD 3301.04  ; AS.GRIPPER UNIT DOWN CONFIRM
AND 3301.05  ; AS.GRIPPER UNIT UP CONFIRM
OR AL83  ; AL83_AS.DIAPH GRIPPER UNIT FAULT
OUT AL83  ; AL83_AS.DIAPH GRIPPER UNIT FAULT
; rung 70
LD 3301.06  ; AS.GRIPPER 1 DIAPH CHUCK. CONFIRM
AND 3301.07  ; AS.GRIPPER 1 DIAPH UNCHUCK. CONFIRM
OR AL84  ; AL84_AS.DIAPH GRIPPER 1 FAULT
OUT AL84  ; AL84_AS.DIAPH GRIPPER 1 FAULT
; rung 71
LD 3301.08  ; AS.GRIPPER 2 DIAPH CHUCK. CONFIRM
AND 3301.09  ; AS.GRIPPER 2 DIAPH UNCHUCK. CONFIRM
OR AL85  ; AL85_AS.DIAPH GRIPPER 2 FAULT
OUT AL85  ; AL85_AS.DIAPH GRIPPER 2 FAULT
; rung 72
LD 3301.10  ; AS.GRIPPER 3 DIAPH CHUCK. CONFIRM
AND 3301.11  ; AS.GRIPPER 3 DIAPH UNCHUCK. CONFIRM
OR AL86  ; AL86_AS.DIAPH GRIPPER 3 FAULT
OUT TR0
AND LT40505
OUT AL86  ; AL86_AS.DIAPH GRIPPER 3 FAULT
LD TR0
TIM LT40505 #5
; rung 73
LD 3301.12  ; AS.FLIP DIAPH 180. CONFIRM
AND 3301.13  ; AS.FLIP DIAPH 0. CONFIRM
OR AL87  ; AL87_AS.DIAPH GRIPPER FLIP FAULT
OUT AL87  ; AL87_AS.DIAPH GRIPPER FLIP FAULT
; rung 74
LD 3302.00  ; AS.GIPPER TRANSFER 1 UNIT CHUCK CONFIRM
AND 3302.01  ; AS.GIPPER TRANSFER 1 UNIT  UNCHUCK CONFIRM
OR AL88  ; AL88_AS.ROTARY GRIPPER 1 FAULT
OUT TR0
AND LT323
OUT AL88  ; AL88_AS.ROTARY GRIPPER 1 FAULT
LD TR0
TIM LT323 #5

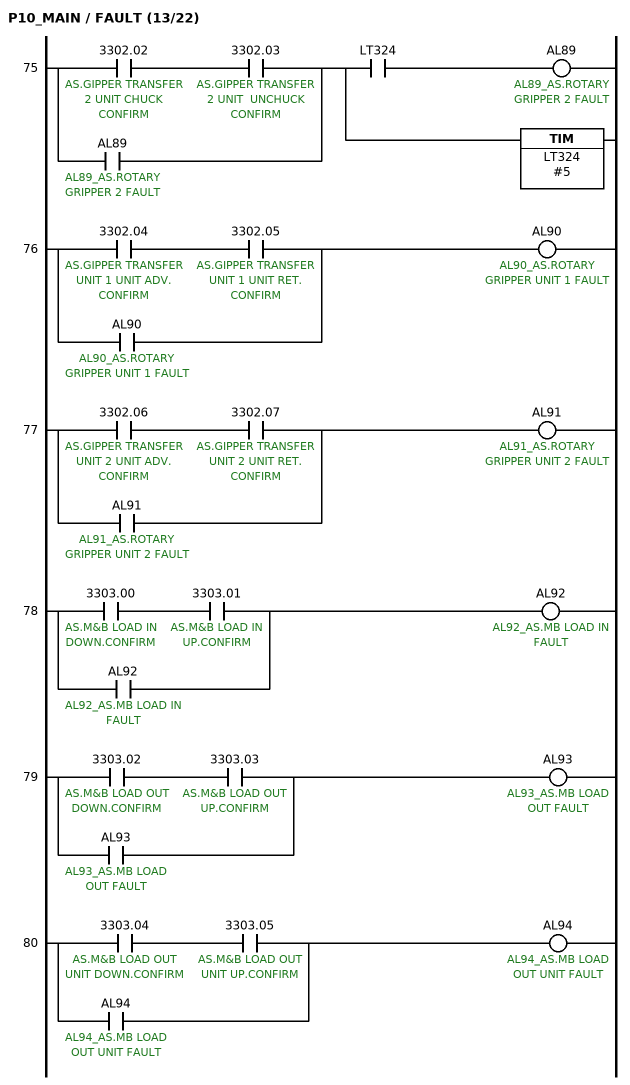
; rung 75
LD 3302.02  ; AS.GIPPER TRANSFER 2 UNIT CHUCK CONFIRM
AND 3302.03  ; AS.GIPPER TRANSFER 2 UNIT  UNCHUCK CONFIRM
OR AL89  ; AL89_AS.ROTARY GRIPPER 2 FAULT
OUT TR0
AND LT324
OUT AL89  ; AL89_AS.ROTARY GRIPPER 2 FAULT
LD TR0
TIM LT324 #5
; rung 76
LD 3302.04  ; AS.GIPPER TRANSFER UNIT 1 UNIT ADV. CONFIRM
AND 3302.05  ; AS.GIPPER TRANSFER UNIT 1 UNIT RET. CONFIRM
OR AL90  ; AL90_AS.ROTARY GRIPPER UNIT 1 FAULT
OUT AL90  ; AL90_AS.ROTARY GRIPPER UNIT 1 FAULT
; rung 77
LD 3302.06  ; AS.GIPPER TRANSFER UNIT 2 UNIT ADV. CONFIRM
AND 3302.07  ; AS.GIPPER TRANSFER UNIT 2 UNIT RET. CONFIRM
OR AL91  ; AL91_AS.ROTARY GRIPPER UNIT 2 FAULT
OUT AL91  ; AL91_AS.ROTARY GRIPPER UNIT 2 FAULT
; rung 78
LD 3303.00  ; AS.M&B LOAD IN DOWN.CONFIRM
AND 3303.01  ; AS.M&B LOAD IN UP.CONFIRM
OR AL92  ; AL92_AS.MB LOAD IN FAULT
OUT AL92  ; AL92_AS.MB LOAD IN FAULT
; rung 79
LD 3303.02  ; AS.M&B LOAD OUT DOWN.CONFIRM
AND 3303.03  ; AS.M&B LOAD OUT UP.CONFIRM
OR AL93  ; AL93_AS.MB LOAD OUT FAULT
OUT AL93  ; AL93_AS.MB LOAD OUT FAULT
; rung 80
LD 3303.04  ; AS.M&B LOAD OUT UNIT DOWN.CONFIRM
AND 3303.05  ; AS.M&B LOAD OUT UNIT UP.CONFIRM
OR AL94  ; AL94_AS.MB LOAD OUT UNIT FAULT
OUT AL94  ; AL94_AS.MB LOAD OUT UNIT FAULT

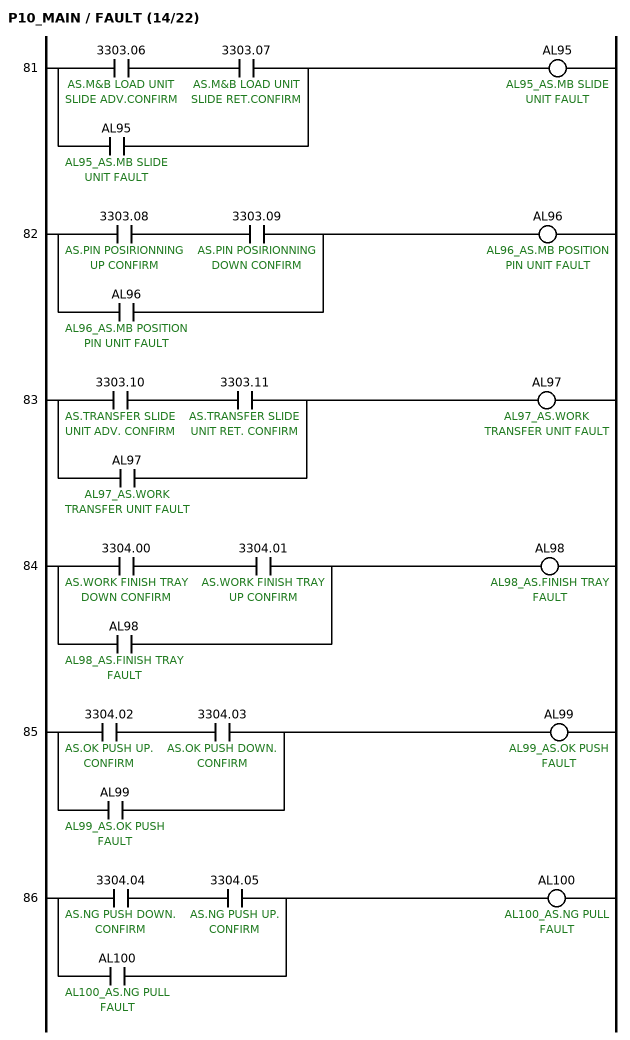
; rung 81
LD 3303.06  ; AS.M&B LOAD UNIT SLIDE ADV.CONFIRM
AND 3303.07  ; AS.M&B LOAD UNIT SLIDE RET.CONFIRM
OR AL95  ; AL95_AS.MB SLIDE UNIT FAULT
OUT AL95  ; AL95_AS.MB SLIDE UNIT FAULT
; rung 82
LD 3303.08  ; AS.PIN POSIRIONNING UP CONFIRM
AND 3303.09  ; AS.PIN POSIRIONNING DOWN CONFIRM
OR AL96  ; AL96_AS.MB POSITION PIN UNIT FAULT
OUT AL96  ; AL96_AS.MB POSITION PIN UNIT FAULT
; rung 83
LD 3303.10  ; AS.TRANSFER SLIDE UNIT ADV. CONFIRM
AND 3303.11  ; AS.TRANSFER SLIDE UNIT RET. CONFIRM
OR AL97  ; AL97_AS.WORK TRANSFER UNIT FAULT
OUT AL97  ; AL97_AS.WORK TRANSFER UNIT FAULT
; rung 84
LD 3304.00  ; AS.WORK FINISH TRAY DOWN CONFIRM
AND 3304.01  ; AS.WORK FINISH TRAY UP CONFIRM
OR AL98  ; AL98_AS.FINISH TRAY FAULT
OUT AL98  ; AL98_AS.FINISH TRAY FAULT
; rung 85
LD 3304.02  ; AS.OK PUSH UP. CONFIRM
AND 3304.03  ; AS.OK PUSH DOWN. CONFIRM
OR AL99  ; AL99_AS.OK PUSH FAULT
OUT AL99  ; AL99_AS.OK PUSH FAULT
; rung 86
LD 3304.04  ; AS.NG PUSH DOWN. CONFIRM
AND 3304.05  ; AS.NG PUSH UP. CONFIRM
OR AL100  ; AL100_AS.NG PULL FAULT
OUT AL100  ; AL100_AS.NG PULL FAULT

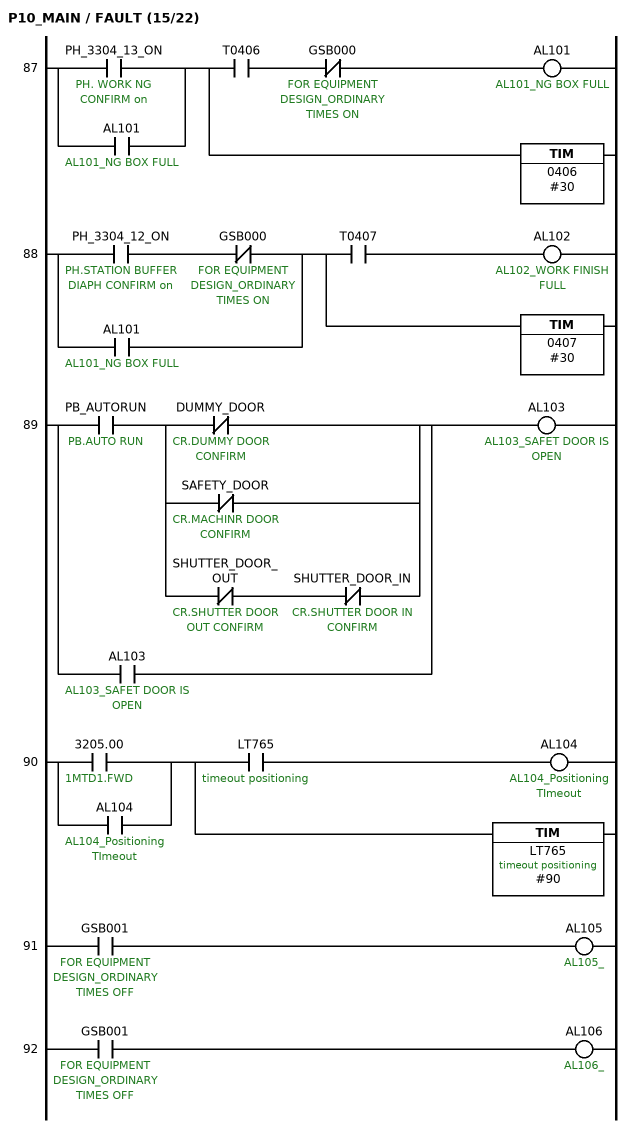
; rung 87
LD PH_3304_13_ON  ; PH. WORK NG CONFIRM on
OR AL101  ; AL101_NG BOX FULL
OUT TR0
AND T0406
ANDNOT GSB000  ; FOR EQUIPMENT DESIGN_ORDINARY TIMES ON
OUT AL101  ; AL101_NG BOX FULL
LD TR0
TIM 0406 #30
; rung 88
LD PH_3304_12_ON  ; PH.STATION BUFFER DIAPH CONFIRM on
ANDNOT GSB000  ; FOR EQUIPMENT DESIGN_ORDINARY TIMES ON
OR AL101  ; AL101_NG BOX FULL
OUT TR0
AND T0407
OUT AL102  ; AL102_WORK FINISH FULL
LD TR0
TIM 0407 #30
; rung 89
LD PB_AUTORUN  ; PB.AUTO RUN
LDNOT DUMMY_DOOR  ; CR.DUMMY DOOR CONFIRM
ORNOT SAFETY_DOOR  ; CR.MACHINR DOOR CONFIRM
LDNOT SHUTTER_DOOR_OUT  ; CR.SHUTTER DOOR OUT CONFIRM
ANDNOT SHUTTER_DOOR_IN  ; CR.SHUTTER DOOR IN CONFIRM
ORLD
ANDLD
OR AL103  ; AL103_SAFET DOOR IS OPEN
OUT AL103  ; AL103_SAFET DOOR IS OPEN
; rung 90
LD 3205.00  ; 1MTD1.FWD
OR AL104  ; AL104_Positioning TImeout
OUT TR0
AND LT765  ; timeout positioning
OUT AL104  ; AL104_Positioning TImeout
LD TR0
TIM LT765 #90  ; timeout positioning
; rung 91
LD GSB001  ; FOR EQUIPMENT DESIGN_ORDINARY TIMES OFF
OUT AL105  ; AL105_
; rung 92
LD GSB001  ; FOR EQUIPMENT DESIGN_ORDINARY TIMES OFF
OUT AL106  ; AL106_

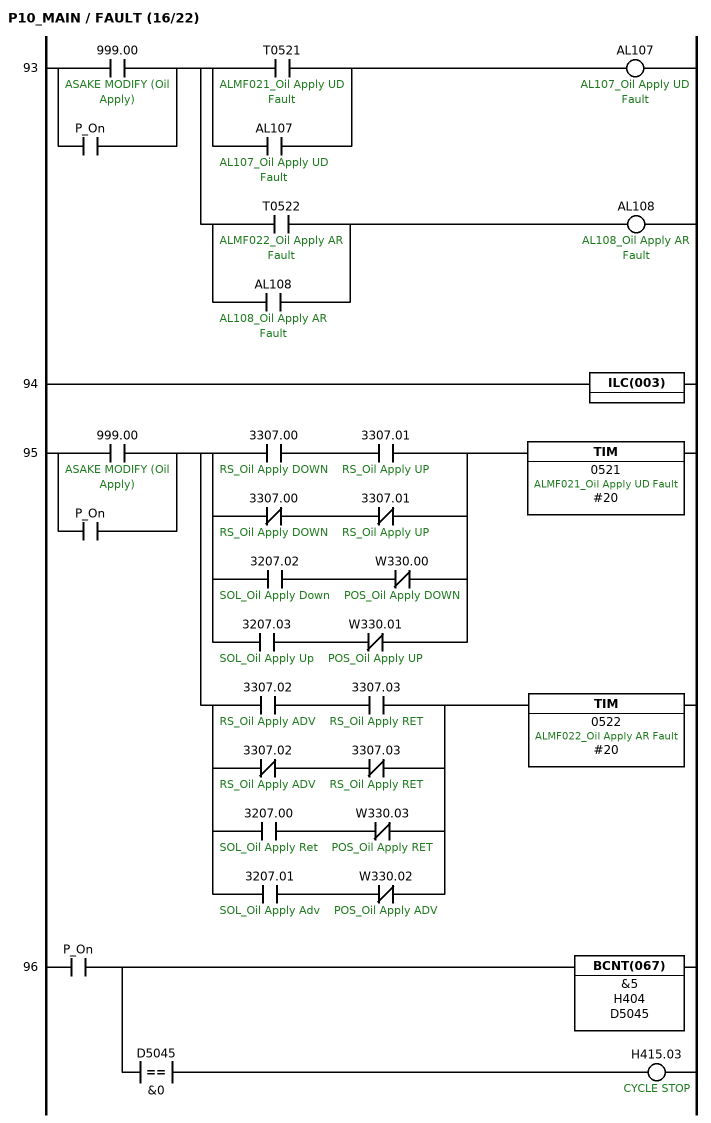
; rung 93
LD 999.00  ; ASAKE MODIFY (Oil Apply)
OR P_On
OUT TR0
LD T0521  ; ALMF021_Oil Apply UD Fault
OR AL107  ; AL107_Oil Apply UD Fault
ANDLD
OUT AL107  ; AL107_Oil Apply UD Fault
LD TR0
LD T0522  ; ALMF022_Oil Apply AR Fault
OR AL108  ; AL108_Oil Apply AR Fault
ANDLD
OUT AL108  ; AL108_Oil Apply AR Fault
; rung 94
ILC(003)
; rung 95
LD 999.00  ; ASAKE MODIFY (Oil Apply)
OR P_On
OUT TR0
LD 3307.00  ; RS_Oil Apply DOWN
AND 3307.01  ; RS_Oil Apply UP
LDNOT 3307.00  ; RS_Oil Apply DOWN
ANDNOT 3307.01  ; RS_Oil Apply UP
ORLD
LD 3207.02  ; SOL_Oil Apply Down
ANDNOT W330.00  ; POS_Oil Apply DOWN
ORLD
LD 3207.03  ; SOL_Oil Apply Up
ANDNOT W330.01  ; POS_Oil Apply UP
ORLD
ANDLD
TIM 0521 #20  ; ALMF021_Oil Apply UD Fault
LD TR0
LD 3307.02  ; RS_Oil Apply ADV
AND 3307.03  ; RS_Oil Apply RET
LDNOT 3307.02  ; RS_Oil Apply ADV
ANDNOT 3307.03  ; RS_Oil Apply RET
ORLD
LD 3207.00  ; SOL_Oil Apply Ret
ANDNOT W330.03  ; POS_Oil Apply RET
ORLD
LD 3207.01  ; SOL_Oil Apply Adv
ANDNOT W330.02  ; POS_Oil Apply ADV
ORLD
ANDLD
TIM 0522 #20  ; ALMF022_Oil Apply AR Fault
; rung 96
LD P_On
BCNT(067) &5 H404 D5045
AND=(300) D5045 &0
OUT H415.03  ; CYCLE STOP

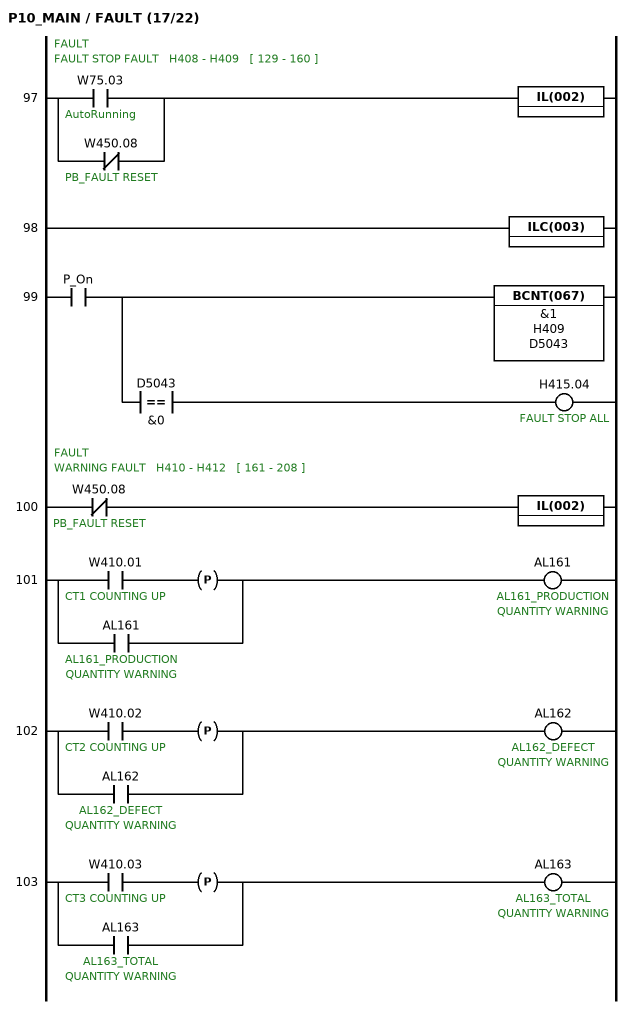
; rung 97: FAULT / FAULT STOP FAULT   H408 - H409   [ 129 - 160 ]
LD W75.03  ; AutoRunning
ORNOT W450.08  ; PB_FAULT RESET
IL(002)
; rung 98
ILC(003)
; rung 99
LD P_On
BCNT(067) &1 H409 D5043
AND=(300) D5043 &0
OUT H415.04  ; FAULT STOP ALL
; rung 100: FAULT / WARNING FAULT   H410 - H412   [ 161 - 208 ]
LDNOT W450.08  ; PB_FAULT RESET
IL(002)
; rung 101
LD W410.01  ; CT1 COUNTING UP
UP(521)
OR AL161  ; AL161_PRODUCTION QUANTITY WARNING
OUT AL161  ; AL161_PRODUCTION QUANTITY WARNING
; rung 102
LD W410.02  ; CT2 COUNTING UP
UP(521)
OR AL162  ; AL162_DEFECT QUANTITY WARNING
OUT AL162  ; AL162_DEFECT QUANTITY WARNING
; rung 103
LD W410.03  ; CT3 COUNTING UP
UP(521)
OR AL163  ; AL163_TOTAL QUANTITY WARNING
OUT AL163  ; AL163_TOTAL QUANTITY WARNING

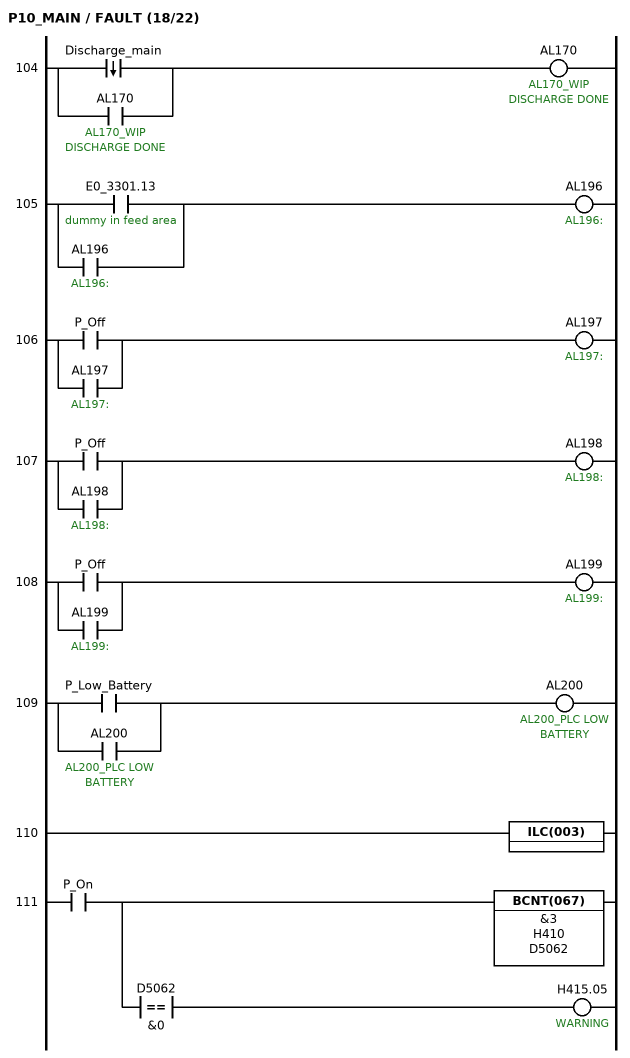
; rung 104
%LD Discharge_main
OR AL170  ; AL170_WIP DISCHARGE DONE
OUT AL170  ; AL170_WIP DISCHARGE DONE
; rung 105
LD E0_3301.13  ; dummy in feed area
OR AL196  ; AL196:
OUT AL196  ; AL196:
; rung 106
LD P_Off
OR AL197  ; AL197:
OUT AL197  ; AL197:
; rung 107
LD P_Off
OR AL198  ; AL198:
OUT AL198  ; AL198:
; rung 108
LD P_Off
OR AL199  ; AL199:
OUT AL199  ; AL199:
; rung 109
LD P_Low_Battery
OR AL200  ; AL200_PLC LOW BATTERY
OUT AL200  ; AL200_PLC LOW BATTERY
; rung 110
ILC(003)
; rung 111
LD P_On
BCNT(067) &3 H410 D5062
AND=(300) D5062 &0
OUT H415.05  ; WARNING

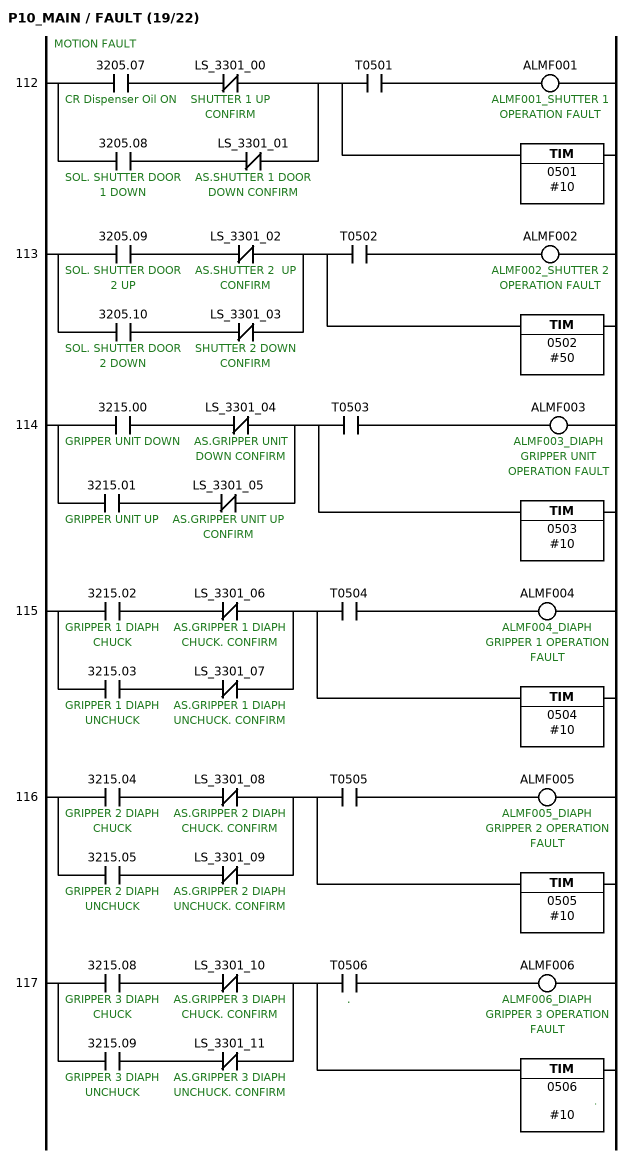
; rung 112: MOTION FAULT
LD 3205.07  ; CR Dispenser Oil ON
ANDNOT LS_3301_00  ; SHUTTER 1 UP CONFIRM
LD 3205.08  ; SOL. SHUTTER DOOR 1 DOWN
ANDNOT LS_3301_01  ; AS.SHUTTER 1 DOOR DOWN CONFIRM
ORLD
OUT TR0
AND T0501
OUT ALMF001  ; ALMF001_SHUTTER 1 OPERATION FAULT
LD TR0
TIM 0501 #10
; rung 113
LD 3205.09  ; SOL. SHUTTER DOOR 2 UP
ANDNOT LS_3301_02  ; AS.SHUTTER 2  UP CONFIRM
LD 3205.10  ; SOL. SHUTTER DOOR 2 DOWN
ANDNOT LS_3301_03  ; SHUTTER 2 DOWN CONFIRM
ORLD
OUT TR0
AND T0502
OUT ALMF002  ; ALMF002_SHUTTER 2 OPERATION FAULT
LD TR0
TIM 0502 #50
; rung 114
LD 3215.00  ; GRIPPER UNIT DOWN
ANDNOT LS_3301_04  ; AS.GRIPPER UNIT DOWN CONFIRM
LD 3215.01  ; GRIPPER UNIT UP
ANDNOT LS_3301_05  ; AS.GRIPPER UNIT UP CONFIRM
ORLD
OUT TR0
AND T0503
OUT ALMF003  ; ALMF003_DIAPH GRIPPER UNIT OPERATION FAULT
LD TR0
TIM 0503 #10
; rung 115
LD 3215.02  ; GRIPPER 1 DIAPH CHUCK
ANDNOT LS_3301_06  ; AS.GRIPPER 1 DIAPH CHUCK. CONFIRM
LD 3215.03  ; GRIPPER 1 DIAPH UNCHUCK
ANDNOT LS_3301_07  ; AS.GRIPPER 1 DIAPH UNCHUCK. CONFIRM
ORLD
OUT TR0
AND T0504
OUT ALMF004  ; ALMF004_DIAPH GRIPPER 1 OPERATION FAULT
LD TR0
TIM 0504 #10
; rung 116
LD 3215.04  ; GRIPPER 2 DIAPH CHUCK
ANDNOT LS_3301_08  ; AS.GRIPPER 2 DIAPH CHUCK. CONFIRM
LD 3215.05  ; GRIPPER 2 DIAPH UNCHUCK
ANDNOT LS_3301_09  ; AS.GRIPPER 2 DIAPH UNCHUCK. CONFIRM
ORLD
OUT TR0
AND T0505
OUT ALMF005  ; ALMF005_DIAPH GRIPPER 2 OPERATION FAULT
LD TR0
TIM 0505 #10
; rung 117
LD 3215.08  ; GRIPPER 3 DIAPH CHUCK
ANDNOT LS_3301_10  ; AS.GRIPPER 3 DIAPH CHUCK. CONFIRM
LD 3215.09  ; GRIPPER 3 DIAPH UNCHUCK
ANDNOT LS_3301_11  ; AS.GRIPPER 3 DIAPH UNCHUCK. CONFIRM
ORLD
OUT TR0
AND T0506  ; .
OUT ALMF006  ; ALMF006_DIAPH GRIPPER 3 OPERATION FAULT
LD TR0
TIM 0506 #10  ; .

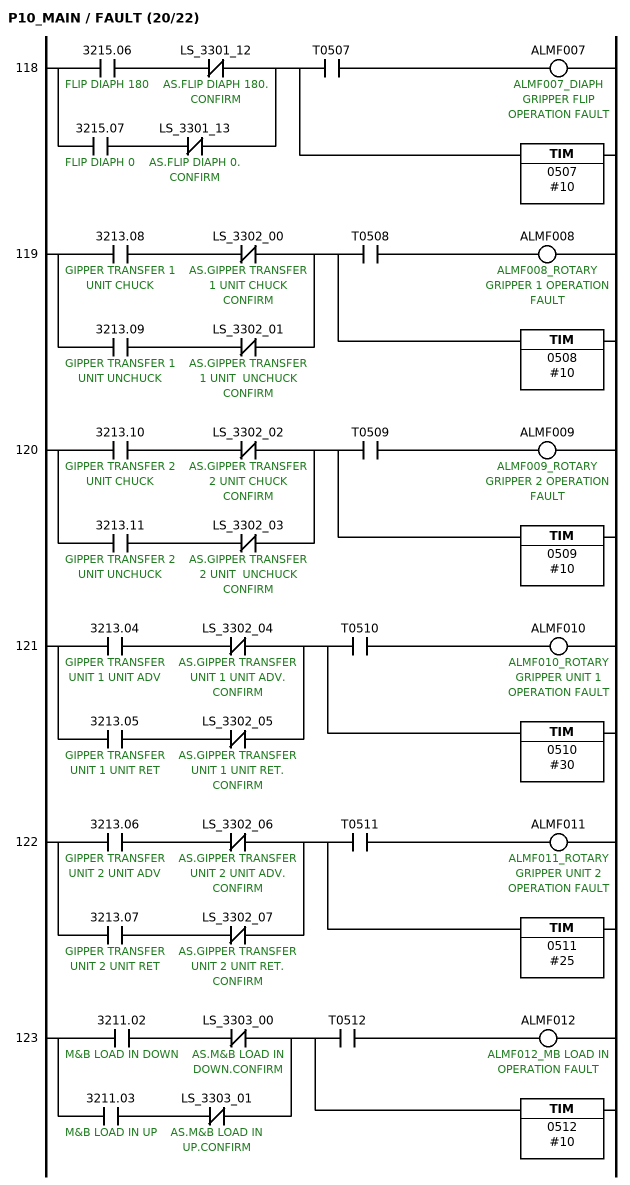
; rung 118
LD 3215.06  ; FLIP DIAPH 180
ANDNOT LS_3301_12  ; AS.FLIP DIAPH 180. CONFIRM
LD 3215.07  ; FLIP DIAPH 0
ANDNOT LS_3301_13  ; AS.FLIP DIAPH 0. CONFIRM
ORLD
OUT TR0
AND T0507
OUT ALMF007  ; ALMF007_DIAPH GRIPPER FLIP OPERATION FAULT
LD TR0
TIM 0507 #10
; rung 119
LD 3213.08  ; GIPPER TRANSFER 1 UNIT CHUCK
ANDNOT LS_3302_00  ; AS.GIPPER TRANSFER 1 UNIT CHUCK CONFIRM
LD 3213.09  ; GIPPER TRANSFER 1 UNIT UNCHUCK
ANDNOT LS_3302_01  ; AS.GIPPER TRANSFER 1 UNIT  UNCHUCK CONFIRM
ORLD
OUT TR0
AND T0508
OUT ALMF008  ; ALMF008_ROTARY GRIPPER 1 OPERATION FAULT
LD TR0
TIM 0508 #10
; rung 120
LD 3213.10  ; GIPPER TRANSFER 2 UNIT CHUCK
ANDNOT LS_3302_02  ; AS.GIPPER TRANSFER 2 UNIT CHUCK CONFIRM
LD 3213.11  ; GIPPER TRANSFER 2 UNIT UNCHUCK
ANDNOT LS_3302_03  ; AS.GIPPER TRANSFER 2 UNIT  UNCHUCK CONFIRM
ORLD
OUT TR0
AND T0509
OUT ALMF009  ; ALMF009_ROTARY GRIPPER 2 OPERATION FAULT
LD TR0
TIM 0509 #10
; rung 121
LD 3213.04  ; GIPPER TRANSFER UNIT 1 UNIT ADV
ANDNOT LS_3302_04  ; AS.GIPPER TRANSFER UNIT 1 UNIT ADV. CONFIRM
LD 3213.05  ; GIPPER TRANSFER UNIT 1 UNIT RET
ANDNOT LS_3302_05  ; AS.GIPPER TRANSFER UNIT 1 UNIT RET. CONFIRM
ORLD
OUT TR0
AND T0510
OUT ALMF010  ; ALMF010_ROTARY GRIPPER UNIT 1 OPERATION FAULT
LD TR0
TIM 0510 #30
; rung 122
LD 3213.06  ; GIPPER TRANSFER UNIT 2 UNIT ADV
ANDNOT LS_3302_06  ; AS.GIPPER TRANSFER UNIT 2 UNIT ADV. CONFIRM
LD 3213.07  ; GIPPER TRANSFER UNIT 2 UNIT RET
ANDNOT LS_3302_07  ; AS.GIPPER TRANSFER UNIT 2 UNIT RET. CONFIRM
ORLD
OUT TR0
AND T0511
OUT ALMF011  ; ALMF011_ROTARY GRIPPER UNIT 2 OPERATION FAULT
LD TR0
TIM 0511 #25
; rung 123
LD 3211.02  ; M&B LOAD IN DOWN
ANDNOT LS_3303_00  ; AS.M&B LOAD IN DOWN.CONFIRM
LD 3211.03  ; M&B LOAD IN UP
ANDNOT LS_3303_01  ; AS.M&B LOAD IN UP.CONFIRM
ORLD
OUT TR0
AND T0512
OUT ALMF012  ; ALMF012_MB LOAD IN OPERATION FAULT
LD TR0
TIM 0512 #10

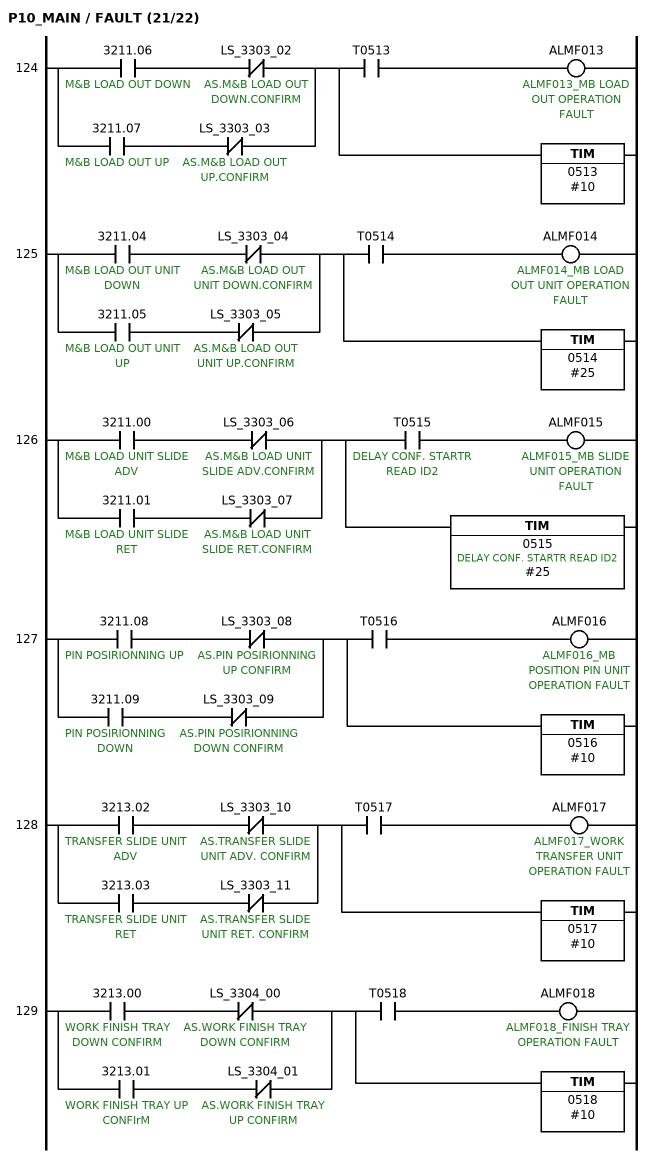
; rung 124
LD 3211.06  ; M&B LOAD OUT DOWN
ANDNOT LS_3303_02  ; AS.M&B LOAD OUT DOWN.CONFIRM
LD 3211.07  ; M&B LOAD OUT UP
ANDNOT LS_3303_03  ; AS.M&B LOAD OUT UP.CONFIRM
ORLD
OUT TR0
AND T0513
OUT ALMF013  ; ALMF013_MB LOAD OUT OPERATION FAULT
LD TR0
TIM 0513 #10
; rung 125
LD 3211.04  ; M&B LOAD OUT UNIT DOWN
ANDNOT LS_3303_04  ; AS.M&B LOAD OUT UNIT DOWN.CONFIRM
LD 3211.05  ; M&B LOAD OUT UNIT UP
ANDNOT LS_3303_05  ; AS.M&B LOAD OUT UNIT UP.CONFIRM
ORLD
OUT TR0
AND T0514
OUT ALMF014  ; ALMF014_MB LOAD OUT UNIT OPERATION FAULT
LD TR0
TIM 0514 #25
; rung 126
LD 3211.00  ; M&B LOAD UNIT SLIDE ADV
ANDNOT LS_3303_06  ; AS.M&B LOAD UNIT SLIDE ADV.CONFIRM
LD 3211.01  ; M&B LOAD UNIT SLIDE RET
ANDNOT LS_3303_07  ; AS.M&B LOAD UNIT SLIDE RET.CONFIRM
ORLD
OUT TR0
AND T0515  ; DELAY CONF. STARTR READ ID2
OUT ALMF015  ; ALMF015_MB SLIDE UNIT OPERATION FAULT
LD TR0
TIM 0515 #25  ; DELAY CONF. STARTR READ ID2
; rung 127
LD 3211.08  ; PIN POSIRIONNING UP
ANDNOT LS_3303_08  ; AS.PIN POSIRIONNING UP CONFIRM
LD 3211.09  ; PIN POSIRIONNING DOWN
ANDNOT LS_3303_09  ; AS.PIN POSIRIONNING DOWN CONFIRM
ORLD
OUT TR0
AND T0516
OUT ALMF016  ; ALMF016_MB POSITION PIN UNIT OPERATION FAULT
LD TR0
TIM 0516 #10
; rung 128
LD 3213.02  ; TRANSFER SLIDE UNIT ADV
ANDNOT LS_3303_10  ; AS.TRANSFER SLIDE UNIT ADV. CONFIRM
LD 3213.03  ; TRANSFER SLIDE UNIT RET
ANDNOT LS_3303_11  ; AS.TRANSFER SLIDE UNIT RET. CONFIRM
ORLD
OUT TR0
AND T0517
OUT ALMF017  ; ALMF017_WORK TRANSFER UNIT OPERATION FAULT
LD TR0
TIM 0517 #10
; rung 129
LD 3213.00  ; WORK FINISH TRAY DOWN CONFIRM
ANDNOT LS_3304_00  ; AS.WORK FINISH TRAY DOWN CONFIRM
LD 3213.01  ; WORK FINISH TRAY UP CONFIrM
ANDNOT LS_3304_01  ; AS.WORK FINISH TRAY UP CONFIRM
ORLD
OUT TR0
AND T0518
OUT ALMF018  ; ALMF018_FINISH TRAY OPERATION FAULT
LD TR0
TIM 0518 #10

